LIN {X 0,Y 509.075,Z 406.145,A -85,B 0,C 180,E1 -5489.209,E2 -5489.209} C_VEL
LIN {X 0,Y 509.075,Z 406.145,A -85,B 0,C 180,E1 -5490.791,E2 -5490.791} C_VEL
LIN {X 0,Y 509.114,Z 405.559,A -85,B 0,C 180,E1 -5491.582,E2 -5491.582} C_VEL
LIN {X 0,Y 509.203,Z 403.121,A -85,B 0,C 180,E1 -5493.165,E2 -5493.165} C_VEL
LIN {X 0,Y 509.209,Z 400.177,A -85,B 0,C 180,E1 -5494.353,E2 -5494.353} C_VEL
LIN {X 0,Y 509.293,Z 396.195,A -85,B 0,C 180,E1 -5495.543,E2 -5495.543} C_VEL
LIN {X 0,Y 509.357,Z 391.927,A -85,B 0,C 180,E1 -5496.557,E2 -5496.557} C_VEL
LIN {X 0,Y 509.449,Z 386.963,A -85,B 0,C 180,E1 -5497.53,E2 -5497.53} C_VEL
LIN {X 0,Y 509.619,Z 380.867,A -85,B 0,C 180,E1 -5498.525,E2 -5498.525} C_VEL
LIN {X 0,Y 509.789,Z 375.167,A -85,B 0,C 180,E1 -5499.322,E2 -5499.322} C_VEL
LIN {X 0,Y 510.017,Z 366.61,A -85,B 0,C 180,E1 -5500.319,E2 -5500.319} C_VEL
LIN {X 0,Y 510.299,Z 358.429,A -85,B 0,C 180,E1 -5501.117,E2 -5501.117} C_VEL
LIN {X 0,Y 510.571,Z 349.915,A -85,B 0,C 180,E1 -5501.815,E2 -5501.815} C_VEL
LIN {X 0,Y 510.752,Z 341.423,A -85,B 0,C 180,E1 -5502.401,E2 -5502.401} C_VEL
LIN {X 0,Y 511.054,Z 331.433,A -85,B 0,C 180,E1 -5502.963,E2 -5502.963} C_VEL
LIN {X 0,Y 511.333,Z 321.35,A -85,B 0,C 180,E1 -5503.411,E2 -5503.411} C_VEL
LIN {X 0,Y 511.369,Z 314.018,A -85,B 0,C 180,E1 -5503.676,E2 -5503.676} C_VEL
LIN {X 0,Y 509.54,Z 302.645,A -85,B 0,C 180,E1 -5504.021,E2 -5504.021} C_VEL
LIN {X 0,Y 509.248,Z 300.709,A -85,B 0,C 180,E1 -5504.077,E2 -5504.077} C_VEL
LIN {X 0,Y 509.293,Z 294.675,A -85,B 0,C 180,E1 -5506.845,E2 -5506.845} C_VEL
LIN {X 0,Y 509.362,Z 289.361,A -85,B 0,C 180,E1 -5509.338,E2 -5509.338} C_VEL
LIN {X 0,Y 509.468,Z 282.918,A -85,B 0,C 180,E1 -5512.441,E2 -5512.441} C_VEL
LIN {X 0,Y 509.557,Z 277.151,A -85,B 0,C 180,E1 -5515.312,E2 -5515.312} C_VEL
LIN {X 0,Y 509.71,Z 271.804,A -85,B 0,C 180,E1 -5518.058,E2 -5518.058} C_VEL
LIN {X 0,Y 509.892,Z 266.964,A -85,B 0,C 180,E1 -5520.662,E2 -5520.662} C_VEL
LIN {X 0,Y 510.073,Z 262.008,A -85,B 0,C 180,E1 -5523.444,E2 -5523.444} C_VEL
LIN {X 0,Y 510.239,Z 257.149,A -85,B 0,C 180,E1 -5526.318,E2 -5526.318} C_VEL
LIN {X 0,Y 510.389,Z 252.423,A -85,B 0,C 180,E1 -5529.301,E2 -5529.301} C_VEL
LIN {X 0,Y 510.459,Z 248.462,A -85,B 0,C 180,E1 -5531.969,E2 -5531.969} C_VEL
LIN {X 0,Y 510.205,Z 245.375,A -85,B 0,C 180,E1 -5534.248,E2 -5534.248} C_VEL
LIN {X 0,Y 509.818,Z 242.618,A -85,B 0,C 180,E1 -5536.425,E2 -5536.425} C_VEL
LIN {X 0,Y 509.825,Z 242.479,A -85,B 0,C 180,E1 -5539.302,E2 -5539.302} C_VEL
LIN {X 0,Y 509.853,Z 242.477,A -85,B 0,C 180,E1 -5541.784,E2 -5541.784} C_VEL
LIN {X 0,Y 509.828,Z 242.479,A -85,B 0,C 180,E1 -5544.619,E2 -5544.619} C_VEL
LIN {X 0,Y 509.864,Z 242.471,A -85,B 0,C 180,E1 -5547.478,E2 -5547.478} C_VEL
LIN {X 0,Y 509.861,Z 242.474,A -85,B 0,C 180,E1 -5550.271,E2 -5550.271} C_VEL
LIN {X 0,Y 509.832,Z 242.473,A -85,B 0,C 180,E1 -5552.938,E2 -5552.938} C_VEL
LIN {X 0,Y 509.845,Z 242.476,A -85,B 0,C 180,E1 -5555.569,E2 -5555.569} C_VEL
LIN {X 0,Y 509.821,Z 242.478,A -85,B 0,C 180,E1 -5558.145,E2 -5558.145} C_VEL
LIN {X 0,Y 509.854,Z 242.47,A -85,B 0,C 180,E1 -5560.678,E2 -5560.678} C_VEL
LIN {X 0,Y 509.861,Z 242.472,A -85,B 0,C 180,E1 -5563.17,E2 -5563.17} C_VEL
LIN {X 0,Y 509.857,Z 242.479,A -85,B 0,C 180,E1 -5565.63,E2 -5565.63} C_VEL
LIN {X 0,Y 509.905,Z 242.465,A -85,B 0,C 180,E1 -5568.87,E2 -5568.87} C_VEL
LIN {X 0,Y 509.905,Z 242.465,A -85,B 0,C 180,E1 -5572.074,E2 -5572.074} C_VEL
LIN {X 0,Y 509.959,Z 242.457,A -85,B 0,C 180,E1 -5574.46,E2 -5574.46} C_VEL
LIN {X 0,Y 510.034,Z 242.452,A -85,B 0,C 180,E1 -5577.626,E2 -5577.626} C_VEL
LIN {X 0,Y 510.038,Z 242.448,A -85,B 0,C 180,E1 -5579.995,E2 -5579.995} C_VEL
LIN {X 0,Y 510.035,Z 242.448,A -85,B 0,C 180,E1 -5582.364,E2 -5582.364} C_VEL
LIN {X 0,Y 509.951,Z 242.461,A -85,B 0,C 180,E1 -5585.531,E2 -5585.531} C_VEL
LIN {X 0,Y 509.902,Z 242.464,A -85,B 0,C 180,E1 -5587.917,E2 -5587.917} C_VEL
LIN {X 0,Y 509.895,Z 242.472,A -85,B 0,C 180,E1 -5591.12,E2 -5591.12} C_VEL
LIN {X 0,Y 509.839,Z 242.474,A -85,B 0,C 180,E1 -5594.361,E2 -5594.361} C_VEL
LIN {X 0,Y 509.849,Z 242.48,A -85,B 0,C 180,E1 -5596.821,E2 -5596.821} C_VEL
LIN {X 0,Y 509.889,Z 242.468,A -85,B 0,C 180,E1 -5600.15,E2 -5600.15} C_VEL
LIN {X 0,Y 509.798,Z 242.477,A -85,B 0,C 180,E1 -5603.558,E2 -5603.558} C_VEL
LIN {X 0,Y 509.878,Z 242.473,A -85,B 0,C 180,E1 -5606.373,E2 -5606.373} C_VEL
LIN {X 0,Y 509.841,Z 242.476,A -85,B 0,C 180,E1 -5608.839,E2 -5608.839} C_VEL
LIN {X 0,Y 509.783,Z 242.479,A -85,B 0,C 180,E1 -5611.585,E2 -5611.585} C_VEL
LIN {X 0,Y 509.814,Z 242.484,A -85,B 0,C 180,E1 -5614.408,E2 -5614.408} C_VEL
LIN {X 0,Y 509.776,Z 242.48,A -85,B 0,C 180,E1 -5617.336,E2 -5617.336} C_VEL
LIN {X 0,Y 509.817,Z 242.482,A -85,B 0,C 180,E1 -5620.375,E2 -5620.375} C_VEL
LIN {X 0,Y 509.809,Z 242.476,A -85,B 0,C 180,E1 -5623.062,E2 -5623.062} C_VEL
LIN {X 0,Y 509.781,Z 242.484,A -85,B 0,C 180,E1 -5625.788,E2 -5625.788} C_VEL
LIN {X 0,Y 509.819,Z 242.477,A -85,B 0,C 180,E1 -5628.572,E2 -5628.572} C_VEL
LIN {X 0,Y 509.806,Z 242.481,A -85,B 0,C 180,E1 -5631.659,E2 -5631.659} C_VEL
LIN {X 0,Y 509.776,Z 242.485,A -85,B 0,C 180,E1 -5633.707,E2 -5633.707} C_VEL
LIN {X 0,Y 509.108,Z 242.566,A -85,B 0,C 180,E1 -5634.367,E2 -5634.367} C_VEL
LIN {X 0,Y 506.292,Z 242.917,A -85,B 0,C 180,E1 -5635.439,E2 -5635.439} C_VEL
LIN {X 0,Y 503.9,Z 243.215,A -85,B 0,C 180,E1 -5636.302,E2 -5636.302} C_VEL
LIN {X 0,Y 502.851,Z 243.343,A -85,B 0,C 180,E1 -5636.968,E2 -5636.968} C_VEL
LIN {X 0,Y 502.753,Z 243.355,A -85,B 0,C 180,E1 -5637.194,E2 -5637.194} C_VEL
LIN {X 0,Y 502.771,Z 243.357,A -85,B 0,C 180,E1 -5640.058,E2 -5640.058} C_VEL
LIN {X 0,Y 502.775,Z 243.352,A -85,B 0,C 180,E1 -5642.531,E2 -5642.531} C_VEL
LIN {X 0,Y 502.781,Z 243.356,A -85,B 0,C 180,E1 -5645.292,E2 -5645.292} C_VEL
LIN {X 0,Y 502.757,Z 243.359,A -85,B 0,C 180,E1 -5647.826,E2 -5647.826} C_VEL
LIN {X 0,Y 502.761,Z 243.354,A -85,B 0,C 180,E1 -5650.398,E2 -5650.398} C_VEL
LIN {X 0,Y 502.783,Z 243.356,A -85,B 0,C 180,E1 -5652.93,E2 -5652.93} C_VEL
LIN {X 0,Y 502.796,Z 243.359,A -85,B 0,C 180,E1 -5655.428,E2 -5655.428} C_VEL
LIN {X 0,Y 502.831,Z 243.349,A -85,B 0,C 180,E1 -5658.716,E2 -5658.716} C_VEL
LIN {X 0,Y 502.851,Z 243.346,A -85,B 0,C 180,E1 -5661.966,E2 -5661.966} C_VEL
LIN {X 0,Y 502.899,Z 243.34,A -85,B 0,C 180,E1 -5664.386,E2 -5664.386} C_VEL
LIN {X 0,Y 502.96,Z 243.333,A -85,B 0,C 180,E1 -5667.598,E2 -5667.598} C_VEL
LIN {X 0,Y 502.955,Z 243.333,A -85,B 0,C 180,E1 -5670,E2 -5670} C_VEL
LIN {X 0,Y 502.96,Z 243.333,A -85,B 0,C 180,E1 -5672.402,E2 -5672.402} C_VEL
LIN {X 0,Y 502.899,Z 243.34,A -85,B 0,C 180,E1 -5675.614,E2 -5675.614} C_VEL
LIN {X 0,Y 502.851,Z 243.346,A -85,B 0,C 180,E1 -5678.034,E2 -5678.034} C_VEL
LIN {X 0,Y 502.831,Z 243.349,A -85,B 0,C 180,E1 -5681.284,E2 -5681.284} C_VEL
LIN {X 0,Y 502.796,Z 243.359,A -85,B 0,C 180,E1 -5684.572,E2 -5684.572} C_VEL
LIN {X 0,Y 502.813,Z 243.351,A -85,B 0,C 180,E1 -5687.908,E2 -5687.908} C_VEL
LIN {X 0,Y 502.766,Z 243.362,A -85,B 0,C 180,E1 -5690.539,E2 -5690.539} C_VEL
LIN {X 0,Y 502.759,Z 243.356,A -85,B 0,C 180,E1 -5693.042,E2 -5693.042} C_VEL
LIN {X 0,Y 502.791,Z 243.351,A -85,B 0,C 180,E1 -5695.678,E2 -5695.678} C_VEL
LIN {X 0,Y 502.783,Z 243.359,A -85,B 0,C 180,E1 -5698.375,E2 -5698.375} C_VEL
LIN {X 0,Y 502.737,Z 243.358,A -85,B 0,C 180,E1 -5701.503,E2 -5701.503} C_VEL
LIN {X 0,Y 502.749,Z 243.36,A -85,B 0,C 180,E1 -5704.448,E2 -5704.448} C_VEL
LIN {X 0,Y 502.726,Z 243.358,A -85,B 0,C 180,E1 -5707.182,E2 -5707.182} C_VEL
LIN {X 0,Y 502.79,Z 243.359,A -85,B 0,C 180,E1 -5710.014,E2 -5710.014} C_VEL
LIN {X 0,Y 502.774,Z 243.357,A -85,B 0,C 180,E1 -5712.206,E2 -5712.206} C_VEL
LIN {X 0,Y 502.766,Z 243.359,A -85,B 0,C 180,E1 -5715.669,E2 -5715.669} C_VEL
LIN {X 0,Y 502.783,Z 243.352,A -85,B 0,C 180,E1 -5718.94,E2 -5718.94} C_VEL
LIN {X 0,Y 502.75,Z 243.359,A -85,B 0,C 180,E1 -5722.051,E2 -5722.051} C_VEL
LIN {X 0,Y 502.769,Z 243.354,A -85,B 0,C 180,E1 -5725.04,E2 -5725.04} C_VEL
LIN {X 0,Y 502.746,Z 243.36,A -85,B 0,C 180,E1 -5727.92,E2 -5727.92} C_VEL
LIN {X 0,Y 502.788,Z 243.351,A -85,B 0,C 180,E1 -5730.717,E2 -5730.717} C_VEL
LIN {X 0,Y 502.829,Z 243.354,A -85,B 0,C 180,E1 -5733.444,E2 -5733.444} C_VEL
LIN {X 0,Y 502.753,Z 243.356,A -85,B 0,C 180,E1 -5736.091,E2 -5736.091} C_VEL
LIN {X 0,Y 502.755,Z 243.356,A -85,B 0,C 180,E1 -5738.694,E2 -5738.694} C_VEL
LIN {X 0,Y 502.8,Z 243.358,A -85,B 0,C 180,E1 -5741.253,E2 -5741.253} C_VEL
LIN {X 0,Y 502.825,Z 243.348,A -85,B 0,C 180,E1 -5744.605,E2 -5744.605} C_VEL
LIN {X 0,Y 502.857,Z 243.342,A -85,B 0,C 180,E1 -5748.043,E2 -5748.043} C_VEL
LIN {X 0,Y 502.844,Z 243.35,A -85,B 0,C 180,E1 -5751.161,E2 -5751.161} C_VEL
LIN {X 0,Y 502.876,Z 243.341,A -85,B 0,C 180,E1 -5753.586,E2 -5753.586} C_VEL
LIN {X 0,Y 502.881,Z 243.347,A -85,B 0,C 180,E1 -5756.8,E2 -5756.8} C_VEL
LIN {X 0,Y 502.999,Z 243.327,A -85,B 0,C 180,E1 -5759.204,E2 -5759.204} C_VEL
LIN {X 0,Y 503.023,Z 243.329,A -85,B 0,C 180,E1 -5760.805,E2 -5760.805} C_VEL
LIN {X 0,Y 502.85,Z 243.345,A -85,B 0,C 180,E1 -5763.209,E2 -5763.209} C_VEL
LIN {X 0,Y 502.884,Z 243.345,A -85,B 0,C 180,E1 -5766.424,E2 -5766.424} C_VEL
LIN {X 0,Y 502.842,Z 243.348,A -85,B 0,C 180,E1 -5768.848,E2 -5768.848} C_VEL
LIN {X 0,Y 502.841,Z 243.348,A -85,B 0,C 180,E1 -5772.106,E2 -5772.106} C_VEL
LIN {X 0,Y 502.846,Z 243.343,A -85,B 0,C 180,E1 -5775.404,E2 -5775.404} C_VEL
LIN {X 0,Y 502.82,Z 243.349,A -85,B 0,C 180,E1 -5778.756,E2 -5778.756} C_VEL
LIN {X 0,Y 502.783,Z 243.351,A -85,B 0,C 180,E1 -5781.315,E2 -5781.315} C_VEL
LIN {X 0,Y 502.773,Z 243.358,A -85,B 0,C 180,E1 -5783.918,E2 -5783.918} C_VEL
LIN {X 0,Y 502.791,Z 243.353,A -85,B 0,C 180,E1 -5786.574,E2 -5786.574} C_VEL
LIN {X 0,Y 502.817,Z 243.355,A -85,B 0,C 180,E1 -5789.938,E2 -5789.938} C_VEL
LIN {X 0,Y 502.834,Z 243.345,A -85,B 0,C 180,E1 -5793.034,E2 -5793.034} C_VEL
LIN {X 0,Y 502.771,Z 243.362,A -85,B 0,C 180,E1 -5795.955,E2 -5795.955} C_VEL
LIN {X 0,Y 502.797,Z 243.354,A -85,B 0,C 180,E1 -5798.98,E2 -5798.98} C_VEL
LIN {X 0,Y 502.782,Z 243.359,A -85,B 0,C 180,E1 -5802.198,E2 -5802.198} C_VEL
LIN {X 0,Y 502.785,Z 243.593,A -85,B 0,C 180,E1 -5803.377,E2 -5803.377} C_VEL
LIN {X 0,Y 503.206,Z 246.497,A -85,B 0,C 180,E1 -5805.709,E2 -5805.709} C_VEL
LIN {X 0,Y 503.444,Z 249.486,A -85,B 0,C 180,E1 -5807.929,E2 -5807.929} C_VEL
LIN {X 0,Y 503.39,Z 252.737,A -85,B 0,C 180,E1 -5810.166,E2 -5810.166} C_VEL
LIN {X 0,Y 503.25,Z 257.244,A -85,B 0,C 180,E1 -5813.095,E2 -5813.095} C_VEL
LIN {X 0,Y 503.074,Z 262.087,A -85,B 0,C 180,E1 -5816.028,E2 -5816.028} C_VEL
LIN {X 0,Y 502.875,Z 266.994,A -85,B 0,C 180,E1 -5818.863,E2 -5818.863} C_VEL
LIN {X 0,Y 502.658,Z 272.27,A -85,B 0,C 180,E1 -5821.748,E2 -5821.748} C_VEL
LIN {X 0,Y 502.499,Z 277.115,A -85,B 0,C 180,E1 -5824.306,E2 -5824.306} C_VEL
LIN {X 0,Y 502.397,Z 282.283,A -85,B 0,C 180,E1 -5826.941,E2 -5826.941} C_VEL
LIN {X 0,Y 502.347,Z 287.694,A -85,B 0,C 180,E1 -5829.615,E2 -5829.615} C_VEL
LIN {X 0,Y 502.22,Z 294.546,A -85,B 0,C 180,E1 -5832.911,E2 -5832.911} C_VEL
LIN {X 0,Y 502.173,Z 300.551,A -85,B 0,C 180,E1 -5835.72,E2 -5835.72} C_VEL
LIN {X 0,Y 504.348,Z 314.257,A -85,B 0,C 180,E1 -5836.143,E2 -5836.143} C_VEL
LIN {X 0,Y 504.491,Z 318.58,A -85,B 0,C 180,E1 -5836.301,E2 -5836.301} C_VEL
LIN {X 0,Y 504.215,Z 329.225,A -85,B 0,C 180,E1 -5836.755,E2 -5836.755} C_VEL
LIN {X 0,Y 503.886,Z 338.977,A -85,B 0,C 180,E1 -5837.286,E2 -5837.286} C_VEL
LIN {X 0,Y 503.647,Z 347.066,A -85,B 0,C 180,E1 -5837.82,E2 -5837.82} C_VEL
LIN {X 0,Y 503.385,Z 355.963,A -85,B 0,C 180,E1 -5838.525,E2 -5838.525} C_VEL
LIN {X 0,Y 503.082,Z 364.495,A -85,B 0,C 180,E1 -5839.333,E2 -5839.333} C_VEL
LIN {X 0,Y 502.86,Z 371.717,A -85,B 0,C 180,E1 -5840.142,E2 -5840.142} C_VEL
LIN {X 0,Y 502.657,Z 377.92,A -85,B 0,C 180,E1 -5840.95,E2 -5840.95} C_VEL
LIN {X 0,Y 502.449,Z 384.456,A -85,B 0,C 180,E1 -5841.96,E2 -5841.96} C_VEL
LIN {X 0,Y 502.339,Z 390.012,A -85,B 0,C 180,E1 -5842.989,E2 -5842.989} C_VEL
LIN {X 0,Y 502.217,Z 394.446,A -85,B 0,C 180,E1 -5843.976,E2 -5843.976} C_VEL
LIN {X 0,Y 502.116,Z 398.766,A -85,B 0,C 180,E1 -5845.183,E2 -5845.183} C_VEL
LIN {X 0,Y 502.141,Z 401.131,A -85,B 0,C 180,E1 -5845.987,E2 -5845.987} C_VEL
LIN {X 0,Y 502.123,Z 402.927,A -85,B 0,C 180,E1 -5846.791,E2 -5846.791} C_VEL
LIN {X 0,Y 502.039,Z 405.365,A -85,B 0,C 180,E1 -5848.396,E2 -5848.396} C_VEL
LIN {X 0,Y 501.992,Z 405.95,A -85,B 0,C 180,E1 -5849.198,E2 -5849.198} C_VEL
LIN {X 0,Y 501.992,Z 405.95,A -85,B 0,C 180,E1 -5850.802,E2 -5850.802} C_VEL
LIN {X 0,Y 502.039,Z 405.365,A -85,B 0,C 180,E1 -5851.604,E2 -5851.604} C_VEL
LIN {X 0,Y 502.123,Z 402.927,A -85,B 0,C 180,E1 -5853.209,E2 -5853.209} C_VEL
LIN {X 0,Y 502.107,Z 399.982,A -85,B 0,C 180,E1 -5854.415,E2 -5854.415} C_VEL
LIN {X 0,Y 502.209,Z 396,A -85,B 0,C 180,E1 -5855.622,E2 -5855.622} C_VEL
LIN {X 0,Y 502.284,Z 391.064,A -85,B 0,C 180,E1 -5856.79,E2 -5856.79} C_VEL
LIN {X 0,Y 502.411,Z 385.612,A -85,B 0,C 180,E1 -5857.839,E2 -5857.839} C_VEL
LIN {X 0,Y 502.593,Z 379.295,A -85,B 0,C 180,E1 -5858.848,E2 -5858.848} C_VEL
LIN {X 0,Y 502.813,Z 373.344,A -85,B 0,C 180,E1 -5859.656,E2 -5859.656} C_VEL
LIN {X 0,Y 502.993,Z 366.415,A -85,B 0,C 180,E1 -5860.465,E2 -5860.465} C_VEL
LIN {X 0,Y 503.291,Z 358.233,A -85,B 0,C 180,E1 -5861.273,E2 -5861.273} C_VEL
LIN {X 0,Y 503.572,Z 349.719,A -85,B 0,C 180,E1 -5861.981,E2 -5861.981} C_VEL
LIN {X 0,Y 503.779,Z 341.832,A -85,B 0,C 180,E1 -5862.538,E2 -5862.538} C_VEL
LIN {X 0,Y 504.112,Z 332.246,A -85,B 0,C 180,E1 -5863.094,E2 -5863.094} C_VEL
LIN {X 0,Y 504.411,Z 322.444,A -85,B 0,C 180,E1 -5863.547,E2 -5863.547} C_VEL
LIN {X 0,Y 504.421,Z 314.697,A -85,B 0,C 180,E1 -5863.842,E2 -5863.842} C_VEL
LIN {X 0,Y 502.472,Z 302.766,A -85,B 0,C 180,E1 -5864.216,E2 -5864.216} C_VEL
LIN {X 0,Y 502.173,Z 300.551,A -85,B 0,C 180,E1 -5864.28,E2 -5864.28} C_VEL
LIN {X 0,Y 502.22,Z 294.542,A -85,B 0,C 180,E1 -5867.089,E2 -5867.089} C_VEL
LIN {X 0,Y 502.344,Z 287.506,A -85,B 0,C 180,E1 -5870.472,E2 -5870.472} C_VEL
LIN {X 0,Y 502.397,Z 282.277,A -85,B 0,C 180,E1 -5873.059,E2 -5873.059} C_VEL
LIN {X 0,Y 502.499,Z 277.109,A -85,B 0,C 180,E1 -5875.694,E2 -5875.694} C_VEL
LIN {X 0,Y 502.666,Z 271.992,A -85,B 0,C 180,E1 -5878.383,E2 -5878.383} C_VEL
LIN {X 0,Y 502.877,Z 266.988,A -85,B 0,C 180,E1 -5881.137,E2 -5881.137} C_VEL
LIN {X 0,Y 503.071,Z 262.038,A -85,B 0,C 180,E1 -5883.972,E2 -5883.972} C_VEL
LIN {X 0,Y 503.252,Z 257.233,A -85,B 0,C 180,E1 -5886.905,E2 -5886.905} C_VEL
LIN {X 0,Y 503.392,Z 252.511,A -85,B 0,C 180,E1 -5889.956,E2 -5889.956} C_VEL
LIN {X 0,Y 503.456,Z 249.175,A -85,B 0,C 180,E1 -5892.278,E2 -5892.278} C_VEL
LIN {X 0,Y 503.154,Z 246.143,A -85,B 0,C 180,E1 -5894.57,E2 -5894.57} C_VEL
LIN {X 0,Y 502.763,Z 243.42,A -85,B 0,C 180,E1 -5896.765,E2 -5896.765} C_VEL
LIN {X 0,Y 502.781,Z 243.357,A -85,B 0,C 180,E1 -5899.009,E2 -5899.009} C_VEL
LIN {X 0,Y 502.794,Z 243.358,A -85,B 0,C 180,E1 -5902.043,E2 -5902.043} C_VEL
LIN {X 0,Y 502.797,Z 243.353,A -85,B 0,C 180,E1 -5905.031,E2 -5905.031} C_VEL
LIN {X 0,Y 502.785,Z 243.358,A -85,B 0,C 180,E1 -5907.912,E2 -5907.912} C_VEL
LIN {X 0,Y 502.814,Z 243.348,A -85,B 0,C 180,E1 -5910.708,E2 -5910.708} C_VEL
LIN {X 0,Y 502.791,Z 243.353,A -85,B 0,C 180,E1 -5913.453,E2 -5913.453} C_VEL
LIN {X 0,Y 502.773,Z 243.358,A -85,B 0,C 180,E1 -5916.082,E2 -5916.082} C_VEL
LIN {X 0,Y 502.783,Z 243.351,A -85,B 0,C 180,E1 -5918.685,E2 -5918.685} C_VEL
LIN {X 0,Y 502.82,Z 243.349,A -85,B 0,C 180,E1 -5921.244,E2 -5921.244} C_VEL
LIN {X 0,Y 502.846,Z 243.343,A -85,B 0,C 180,E1 -5924.596,E2 -5924.596} C_VEL
LIN {X 0,Y 502.873,Z 243.342,A -85,B 0,C 180,E1 -5928.035,E2 -5928.035} C_VEL
LIN {X 0,Y 502.842,Z 243.348,A -85,B 0,C 180,E1 -5931.152,E2 -5931.152} C_VEL
LIN {X 0,Y 502.884,Z 243.345,A -85,B 0,C 180,E1 -5933.576,E2 -5933.576} C_VEL
LIN {X 0,Y 502.85,Z 243.345,A -85,B 0,C 180,E1 -5936.791,E2 -5936.791} C_VEL
LIN {X 0,Y 503.023,Z 243.329,A -85,B 0,C 180,E1 -5939.195,E2 -5939.195} C_VEL
LIN {X 0,Y 503.005,Z 243.324,A -85,B 0,C 180,E1 -5942.397,E2 -5942.397} C_VEL
LIN {X 0,Y 502.905,Z 243.338,A -85,B 0,C 180,E1 -5945.609,E2 -5945.609} C_VEL
LIN {X 0,Y 502.862,Z 243.341,A -85,B 0,C 180,E1 -5948.029,E2 -5948.029} C_VEL
LIN {X 0,Y 502.859,Z 243.346,A -85,B 0,C 180,E1 -5951.278,E2 -5951.278} C_VEL
LIN {X 0,Y 502.82,Z 243.351,A -85,B 0,C 180,E1 -5954.566,E2 -5954.566} C_VEL
LIN {X 0,Y 502.796,Z 243.35,A -85,B 0,C 180,E1 -5957.903,E2 -5957.903} C_VEL
LIN {X 0,Y 502.801,Z 243.355,A -85,B 0,C 180,E1 -5960.531,E2 -5960.531} C_VEL
LIN {X 0,Y 502.76,Z 243.358,A -85,B 0,C 180,E1 -5963.035,E2 -5963.035} C_VEL
LIN {X 0,Y 502.806,Z 243.348,A -85,B 0,C 180,E1 -5965.671,E2 -5965.671} C_VEL
LIN {X 0,Y 502.805,Z 243.355,A -85,B 0,C 180,E1 -5968.368,E2 -5968.368} C_VEL
LIN {X 0,Y 502.755,Z 243.355,A -85,B 0,C 180,E1 -5971.494,E2 -5971.494} C_VEL
LIN {X 0,Y 502.766,Z 243.361,A -85,B 0,C 180,E1 -5974.44,E2 -5974.44} C_VEL
LIN {X 0,Y 502.738,Z 243.357,A -85,B 0,C 180,E1 -5977.174,E2 -5977.174} C_VEL
LIN {X 0,Y 502.776,Z 243.357,A -85,B 0,C 180,E1 -5980.007,E2 -5980.007} C_VEL
LIN {X 0,Y 502.782,Z 243.36,A -85,B 0,C 180,E1 -5982.198,E2 -5982.198} C_VEL
LIN {X 0,Y 502.751,Z 243.356,A -85,B 0,C 180,E1 -5985.464,E2 -5985.464} C_VEL
LIN {X 0,Y 502.786,Z 243.357,A -85,B 0,C 180,E1 -5987.861,E2 -5987.861} C_VEL
LIN {X 0,Y 502.775,Z 243.352,A -85,B 0,C 180,E1 -5991.023,E2 -5991.023} C_VEL
LIN {X 0,Y 502.729,Z 243.363,A -85,B 0,C 180,E1 -5994.164,E2 -5994.164} C_VEL
LIN {X 0,Y 502.753,Z 243.355,A -85,B 0,C 180,E1 -5997.194,E2 -5997.194} C_VEL
LIN {X 0,Y 502.053,Z 243.45,A -85,B 0,C 180,E1 -5997.863,E2 -5997.863} C_VEL
LIN {X 0,Y 499.195,Z 243.8,A -85,B 0,C 180,E1 -5998.949,E2 -5998.949} C_VEL
LIN {X 0,Y 496.804,Z 244.104,A -85,B 0,C 180,E1 -5999.824,E2 -5999.824} C_VEL
LIN {X 0,Y 495.785,Z 244.224,A -85,B 0,C 180,E1 -6000.5,E2 -6000.5} C_VEL
LIN {X 0,Y 495.705,Z 244.233,A -85,B 0,C 180,E1 -6000.728,E2 -6000.728} C_VEL
LIN {X 0,Y 495.744,Z 244.233,A -85,B 0,C 180,E1 -6003.93,E2 -6003.93} C_VEL
LIN {X 0,Y 495.726,Z 244.233,A -85,B 0,C 180,E1 -6007.128,E2 -6007.128} C_VEL
LIN {X 0,Y 495.713,Z 244.234,A -85,B 0,C 180,E1 -6010.108,E2 -6010.108} C_VEL
LIN {X 0,Y 495.736,Z 244.232,A -85,B 0,C 180,E1 -6012.68,E2 -6012.68} C_VEL
LIN {X 0,Y 495.749,Z 244.235,A -85,B 0,C 180,E1 -6015.216,E2 -6015.216} C_VEL
LIN {X 0,Y 495.81,Z 244.222,A -85,B 0,C 180,E1 -6018.554,E2 -6018.554} C_VEL
LIN {X 0,Y 495.819,Z 244.223,A -85,B 0,C 180,E1 -6021.851,E2 -6021.851} C_VEL
LIN {X 0,Y 495.854,Z 244.217,A -85,B 0,C 180,E1 -6024.306,E2 -6024.306} C_VEL
LIN {X 0,Y 495.93,Z 244.209,A -85,B 0,C 180,E1 -6027.563,E2 -6027.563} C_VEL
LIN {X 0,Y 495.926,Z 244.209,A -85,B 0,C 180,E1 -6030,E2 -6030} C_VEL
LIN {X 0,Y 495.93,Z 244.209,A -85,B 0,C 180,E1 -6032.437,E2 -6032.437} C_VEL
LIN {X 0,Y 495.854,Z 244.217,A -85,B 0,C 180,E1 -6035.694,E2 -6035.694} C_VEL
LIN {X 0,Y 495.819,Z 244.223,A -85,B 0,C 180,E1 -6038.149,E2 -6038.149} C_VEL
LIN {X 0,Y 495.81,Z 244.222,A -85,B 0,C 180,E1 -6041.446,E2 -6041.446} C_VEL
LIN {X 0,Y 495.749,Z 244.235,A -85,B 0,C 180,E1 -6044.784,E2 -6044.784} C_VEL
LIN {X 0,Y 495.765,Z 244.232,A -85,B 0,C 180,E1 -6048.258,E2 -6048.258} C_VEL
LIN {X 0,Y 495.702,Z 244.234,A -85,B 0,C 180,E1 -6051.63,E2 -6051.63} C_VEL
LIN {X 0,Y 495.745,Z 244.23,A -85,B 0,C 180,E1 -6054.884,E2 -6054.884} C_VEL
LIN {X 0,Y 495.759,Z 244.227,A -85,B 0,C 180,E1 -6056.977,E2 -6056.977} C_VEL
LIN {X 0,Y 495.717,Z 244.239,A -85,B 0,C 180,E1 -6060.153,E2 -6060.153} C_VEL
LIN {X 0,Y 495.735,Z 244.229,A -85,B 0,C 180,E1 -6063.248,E2 -6063.248} C_VEL
LIN {X 0,Y 495.672,Z 244.246,A -85,B 0,C 180,E1 -6066.094,E2 -6066.094} C_VEL
LIN {X 0,Y 495.732,Z 244.23,A -85,B 0,C 180,E1 -6068.776,E2 -6068.776} C_VEL
LIN {X 0,Y 495.733,Z 244.235,A -85,B 0,C 180,E1 -6071.782,E2 -6071.782} C_VEL
LIN {X 0,Y 495.709,Z 244.233,A -85,B 0,C 180,E1 -6075.143,E2 -6075.143} C_VEL
LIN {X 0,Y 495.739,Z 244.232,A -85,B 0,C 180,E1 -6078.227,E2 -6078.227} C_VEL
LIN {X 0,Y 495.724,Z 244.233,A -85,B 0,C 180,E1 -6081.236,E2 -6081.236} C_VEL
LIN {X 0,Y 495.716,Z 244.232,A -85,B 0,C 180,E1 -6084.468,E2 -6084.468} C_VEL
LIN {X 0,Y 495.729,Z 244.236,A -85,B 0,C 180,E1 -6087.411,E2 -6087.411} C_VEL
LIN {X 0,Y 495.73,Z 244.23,A -85,B 0,C 180,E1 -6090.259,E2 -6090.259} C_VEL
LIN {X 0,Y 495.79,Z 244.229,A -85,B 0,C 180,E1 -6093.256,E2 -6093.256} C_VEL
LIN {X 0,Y 495.716,Z 244.235,A -85,B 0,C 180,E1 -6095.73,E2 -6095.73} C_VEL
LIN {X 0,Y 495.713,Z 244.232,A -85,B 0,C 180,E1 -6098.376,E2 -6098.376} C_VEL
LIN {X 0,Y 495.756,Z 244.232,A -85,B 0,C 180,E1 -6100.977,E2 -6100.977} C_VEL
LIN {X 0,Y 495.783,Z 244.224,A -85,B 0,C 180,E1 -6104.381,E2 -6104.381} C_VEL
LIN {X 0,Y 495.76,Z 244.232,A -85,B 0,C 180,E1 -6106.896,E2 -6106.896} C_VEL
LIN {X 0,Y 495.755,Z 244.23,A -85,B 0,C 180,E1 -6109.386,E2 -6109.386} C_VEL
LIN {X 0,Y 495.818,Z 244.219,A -85,B 0,C 180,E1 -6111.856,E2 -6111.856} C_VEL
LIN {X 0,Y 495.861,Z 244.215,A -85,B 0,C 180,E1 -6114.311,E2 -6114.311} C_VEL
LIN {X 0,Y 495.975,Z 244.2,A -85,B 0,C 180,E1 -6117.569,E2 -6117.569} C_VEL
LIN {X 0,Y 495.972,Z 244.207,A -85,B 0,C 180,E1 -6120.817,E2 -6120.817} C_VEL
LIN {X 0,Y 495.971,Z 244.205,A -85,B 0,C 180,E1 -6122.441,E2 -6122.441} C_VEL
LIN {X 0,Y 495.87,Z 244.213,A -85,B 0,C 180,E1 -6125.698,E2 -6125.698} C_VEL
LIN {X 0,Y 495.822,Z 244.222,A -85,B 0,C 180,E1 -6128.153,E2 -6128.153} C_VEL
LIN {X 0,Y 495.846,Z 244.215,A -85,B 0,C 180,E1 -6131.449,E2 -6131.449} C_VEL
LIN {X 0,Y 495.785,Z 244.226,A -85,B 0,C 180,E1 -6134.787,E2 -6134.787} C_VEL
LIN {X 0,Y 495.778,Z 244.231,A -85,B 0,C 180,E1 -6138.175,E2 -6138.175} C_VEL
LIN {X 0,Y 495.775,Z 244.226,A -85,B 0,C 180,E1 -6140.76,E2 -6140.76} C_VEL
LIN {X 0,Y 495.742,Z 244.229,A -85,B 0,C 180,E1 -6143.391,E2 -6143.391} C_VEL
LIN {X 0,Y 495.745,Z 244.229,A -85,B 0,C 180,E1 -6146.734,E2 -6146.734} C_VEL
LIN {X 0,Y 495.765,Z 244.23,A -85,B 0,C 180,E1 -6149.75,E2 -6149.75} C_VEL
LIN {X 0,Y 495.77,Z 244.226,A -85,B 0,C 180,E1 -6152.598,E2 -6152.598} C_VEL
LIN {X 0,Y 495.747,Z 244.232,A -85,B 0,C 180,E1 -6155.541,E2 -6155.541} C_VEL
LIN {X 0,Y 495.762,Z 244.23,A -85,B 0,C 180,E1 -6158.77,E2 -6158.77} C_VEL
LIN {X 0,Y 495.751,Z 244.236,A -85,B 0,C 180,E1 -6161.785,E2 -6161.785} C_VEL
LIN {X 0,Y 495.715,Z 244.239,A -85,B 0,C 180,E1 -6162.887,E2 -6162.887} C_VEL
LIN {X 0,Y 496.27,Z 248.129,A -85,B 0,C 180,E1 -6166.06,E2 -6166.06} C_VEL
LIN {X 0,Y 496.448,Z 251.591,A -85,B 0,C 180,E1 -6168.619,E2 -6168.619} C_VEL
LIN {X 0,Y 496.294,Z 255.743,A -85,B 0,C 180,E1 -6171.46,E2 -6171.46} C_VEL
LIN {X 0,Y 496.135,Z 260.505,A -85,B 0,C 180,E1 -6174.495,E2 -6174.495} C_VEL
LIN {X 0,Y 495.928,Z 265.372,A -85,B 0,C 180,E1 -6177.418,E2 -6177.418} C_VEL
LIN {X 0,Y 495.731,Z 270.324,A -85,B 0,C 180,E1 -6180.252,E2 -6180.252} C_VEL
LIN {X 0,Y 495.517,Z 275.965,A -85,B 0,C 180,E1 -6183.325,E2 -6183.325} C_VEL
LIN {X 0,Y 495.387,Z 280.503,A -85,B 0,C 180,E1 -6185.707,E2 -6185.707} C_VEL
LIN {X 0,Y 495.278,Z 285.676,A -85,B 0,C 180,E1 -6188.35,E2 -6188.35} C_VEL
LIN {X 0,Y 495.178,Z 290.91,A -85,B 0,C 180,E1 -6190.948,E2 -6190.948} C_VEL
LIN {X 0,Y 495.104,Z 296.196,A -85,B 0,C 180,E1 -6193.507,E2 -6193.507} C_VEL
LIN {X 0,Y 495.063,Z 300.421,A -85,B 0,C 180,E1 -6195.524,E2 -6195.524} C_VEL
LIN {X 0,Y 496.766,Z 310.981,A -85,B 0,C 180,E1 -6195.836,E2 -6195.836} C_VEL
LIN {X 0,Y 497.647,Z 317.097,A -85,B 0,C 180,E1 -6196.057,E2 -6196.057} C_VEL
LIN {X 0,Y 497.316,Z 328.022,A -85,B 0,C 180,E1 -6196.516,E2 -6196.516} C_VEL
LIN {X 0,Y 496.94,Z 339.052,A -85,B 0,C 180,E1 -6197.122,E2 -6197.122} C_VEL
LIN {X 0,Y 496.632,Z 348.171,A -85,B 0,C 180,E1 -6197.745,E2 -6197.745} C_VEL
LIN {X 0,Y 496.361,Z 356.903,A -85,B 0,C 180,E1 -6198.464,E2 -6198.464} C_VEL
LIN {X 0,Y 496.09,Z 364.3,A -85,B 0,C 180,E1 -6199.181,E2 -6199.181} C_VEL
LIN {X 0,Y 495.83,Z 371.521,A -85,B 0,C 180,E1 -6200.001,E2 -6200.001} C_VEL
LIN {X 0,Y 495.624,Z 377.724,A -85,B 0,C 180,E1 -6200.821,E2 -6200.821} C_VEL
LIN {X 0,Y 495.394,Z 384.261,A -85,B 0,C 180,E1 -6201.844,E2 -6201.844} C_VEL
LIN {X 0,Y 495.275,Z 388.762,A -85,B 0,C 180,E1 -6202.663,E2 -6202.663} C_VEL
LIN {X 0,Y 495.13,Z 393.772,A -85,B 0,C 180,E1 -6203.763,E2 -6203.763} C_VEL
LIN {X 0,Y 495.11,Z 397.334,A -85,B 0,C 180,E1 -6204.706,E2 -6204.706} C_VEL
LIN {X 0,Y 495.035,Z 400.936,A -85,B 0,C 180,E1 -6205.93,E2 -6205.93} C_VEL
LIN {X 0,Y 495.045,Z 402.732,A -85,B 0,C 180,E1 -6206.745,E2 -6206.745} C_VEL
LIN {X 0,Y 494.965,Z 405.171,A -85,B 0,C 180,E1 -6208.373,E2 -6208.373} C_VEL
LIN {X 0,Y 494.913,Z 405.756,A -85,B 0,C 180,E1 -6209.186,E2 -6209.186} C_VEL
LIN {X 0,Y 494.913,Z 405.756,A -85,B 0,C 180,E1 -6210.814,E2 -6210.814} C_VEL
LIN {X 0,Y 494.965,Z 405.171,A -85,B 0,C 180,E1 -6211.627,E2 -6211.627} C_VEL
LIN {X 0,Y 495.045,Z 402.732,A -85,B 0,C 180,E1 -6213.255,E2 -6213.255} C_VEL
LIN {X 0,Y 495.014,Z 399.787,A -85,B 0,C 180,E1 -6214.478,E2 -6214.478} C_VEL
LIN {X 0,Y 495.126,Z 395.804,A -85,B 0,C 180,E1 -6215.702,E2 -6215.702} C_VEL
LIN {X 0,Y 495.226,Z 390.678,A -85,B 0,C 180,E1 -6216.928,E2 -6216.928} C_VEL
LIN {X 0,Y 495.352,Z 385.416,A -85,B 0,C 180,E1 -6217.951,E2 -6217.951} C_VEL
LIN {X 0,Y 495.566,Z 379.1,A -85,B 0,C 180,E1 -6218.975,E2 -6218.975} C_VEL
LIN {X 0,Y 495.764,Z 373.148,A -85,B 0,C 180,E1 -6219.794,E2 -6219.794} C_VEL
LIN {X 0,Y 495.987,Z 366.219,A -85,B 0,C 180,E1 -6220.615,E2 -6220.615} C_VEL
LIN {X 0,Y 496.317,Z 358.038,A -85,B 0,C 180,E1 -6221.434,E2 -6221.434} C_VEL
LIN {X 0,Y 496.606,Z 349.524,A -85,B 0,C 180,E1 -6222.152,E2 -6222.152} C_VEL
LIN {X 0,Y 496.886,Z 340.643,A -85,B 0,C 180,E1 -6222.778,E2 -6222.778} C_VEL
LIN {X 0,Y 497.151,Z 331.042,A -85,B 0,C 180,E1 -6223.332,E2 -6223.332} C_VEL
LIN {X 0,Y 497.493,Z 322.249,A -85,B 0,C 180,E1 -6223.739,E2 -6223.739} C_VEL
LIN {X 0,Y 497.466,Z 315.346,A -85,B 0,C 180,E1 -6224.013,E2 -6224.013} C_VEL
LIN {X 0,Y 495.411,Z 302.577,A -85,B 0,C 180,E1 -6224.423,E2 -6224.423} C_VEL
LIN {X 0,Y 495.049,Z 300.392,A -85,B 0,C 180,E1 -6224.49,E2 -6224.49} C_VEL
LIN {X 0,Y 495.162,Z 294.41,A -85,B 0,C 180,E1 -6227.341,E2 -6227.341} C_VEL
LIN {X 0,Y 495.256,Z 287.407,A -85,B 0,C 180,E1 -6230.779,E2 -6230.779} C_VEL
LIN {X 0,Y 495.327,Z 282.205,A -85,B 0,C 180,E1 -6233.408,E2 -6233.408} C_VEL
LIN {X 0,Y 495.452,Z 277.066,A -85,B 0,C 180,E1 -6236.086,E2 -6236.086} C_VEL
LIN {X 0,Y 495.649,Z 271.992,A -85,B 0,C 180,E1 -6238.822,E2 -6238.822} C_VEL
LIN {X 0,Y 495.871,Z 266.785,A -85,B 0,C 180,E1 -6241.743,E2 -6241.743} C_VEL
LIN {X 0,Y 496.079,Z 261.723,A -85,B 0,C 180,E1 -6244.742,E2 -6244.742} C_VEL
LIN {X 0,Y 496.271,Z 257.28,A -85,B 0,C 180,E1 -6247.525,E2 -6247.525} C_VEL
LIN {X 0,Y 496.398,Z 252.625,A -85,B 0,C 180,E1 -6250.636,E2 -6250.636} C_VEL
LIN {X 0,Y 496.4,Z 249.605,A -85,B 0,C 180,E1 -6252.81,E2 -6252.81} C_VEL
LIN {X 0,Y 496.062,Z 246.645,A -85,B 0,C 180,E1 -6255.102,E2 -6255.102} C_VEL
LIN {X 0,Y 495.715,Z 244.239,A -85,B 0,C 180,E1 -6257.113,E2 -6257.113} C_VEL
LIN {X 0,Y 495.75,Z 244.235,A -85,B 0,C 180,E1 -6259.953,E2 -6259.953} C_VEL
LIN {X 0,Y 495.722,Z 244.238,A -85,B 0,C 180,E1 -6262.552,E2 -6262.552} C_VEL
LIN {X 0,Y 495.774,Z 244.229,A -85,B 0,C 180,E1 -6265.453,E2 -6265.453} C_VEL
LIN {X 0,Y 495.757,Z 244.23,A -85,B 0,C 180,E1 -6268.361,E2 -6268.361} C_VEL
LIN {X 0,Y 495.735,Z 244.23,A -85,B 0,C 180,E1 -6271.179,E2 -6271.179} C_VEL
LIN {X 0,Y 495.733,Z 244.238,A -85,B 0,C 180,E1 -6273.925,E2 -6273.925} C_VEL
LIN {X 0,Y 495.759,Z 244.227,A -85,B 0,C 180,E1 -6277.136,E2 -6277.136} C_VEL
LIN {X 0,Y 495.767,Z 244.229,A -85,B 0,C 180,E1 -6280.106,E2 -6280.106} C_VEL
LIN {X 0,Y 495.754,Z 244.227,A -85,B 0,C 180,E1 -6282.676,E2 -6282.676} C_VEL
LIN {X 0,Y 495.785,Z 244.226,A -85,B 0,C 180,E1 -6285.213,E2 -6285.213} C_VEL
LIN {X 0,Y 495.845,Z 244.215,A -85,B 0,C 180,E1 -6288.551,E2 -6288.551} C_VEL
LIN {X 0,Y 495.822,Z 244.221,A -85,B 0,C 180,E1 -6291.847,E2 -6291.847} C_VEL
LIN {X 0,Y 495.87,Z 244.213,A -85,B 0,C 180,E1 -6294.302,E2 -6294.302} C_VEL
LIN {X 0,Y 495.971,Z 244.205,A -85,B 0,C 180,E1 -6297.559,E2 -6297.559} C_VEL
LIN {X 0,Y 495.981,Z 244.199,A -85,B 0,C 180,E1 -6299.995,E2 -6299.995} C_VEL
LIN {X 0,Y 495.975,Z 244.2,A -85,B 0,C 180,E1 -6302.431,E2 -6302.431} C_VEL
LIN {X 0,Y 495.861,Z 244.215,A -85,B 0,C 180,E1 -6305.689,E2 -6305.689} C_VEL
LIN {X 0,Y 495.818,Z 244.219,A -85,B 0,C 180,E1 -6308.144,E2 -6308.144} C_VEL
LIN {X 0,Y 495.833,Z 244.219,A -85,B 0,C 180,E1 -6311.44,E2 -6311.44} C_VEL
LIN {X 0,Y 495.766,Z 244.233,A -85,B 0,C 180,E1 -6314.778,E2 -6314.778} C_VEL
LIN {X 0,Y 495.739,Z 244.231,A -85,B 0,C 180,E1 -6317.314,E2 -6317.314} C_VEL
LIN {X 0,Y 495.743,Z 244.228,A -85,B 0,C 180,E1 -6319.885,E2 -6319.885} C_VEL
LIN {X 0,Y 495.729,Z 244.236,A -85,B 0,C 180,E1 -6322.855,E2 -6322.855} C_VEL
LIN {X 0,Y 495.757,Z 244.229,A -85,B 0,C 180,E1 -6326.063,E2 -6326.063} C_VEL
LIN {X 0,Y 495.737,Z 244.234,A -85,B 0,C 180,E1 -6328.81,E2 -6328.81} C_VEL
LIN {X 0,Y 495.717,Z 244.232,A -85,B 0,C 180,E1 -6331.72,E2 -6331.72} C_VEL
LIN {X 0,Y 495.736,Z 244.233,A -85,B 0,C 180,E1 -6334.69,E2 -6334.69} C_VEL
LIN {X 0,Y 495.688,Z 244.236,A -85,B 0,C 180,E1 -6337.557,E2 -6337.557} C_VEL
LIN {X 0,Y 495.735,Z 244.232,A -85,B 0,C 180,E1 -6340.694,E2 -6340.694} C_VEL
LIN {X 0,Y 495.728,Z 244.233,A -85,B 0,C 180,E1 -6343.696,E2 -6343.696} C_VEL
LIN {X 0,Y 495.712,Z 244.232,A -85,B 0,C 180,E1 -6347.117,E2 -6347.117} C_VEL
LIN {X 0,Y 495.749,Z 244.231,A -85,B 0,C 180,E1 -6350.363,E2 -6350.363} C_VEL
LIN {X 0,Y 495.677,Z 244.239,A -85,B 0,C 180,E1 -6353.453,E2 -6353.453} C_VEL
LIN {X 0,Y 495.703,Z 244.235,A -85,B 0,C 180,E1 -6356.432,E2 -6356.432} C_VEL
LIN {X 0,Y 495.697,Z 244.237,A -85,B 0,C 180,E1 -6359.31,E2 -6359.31} C_VEL
LIN {X 0,Y 495.705,Z 244.233,A -85,B 0,C 180,E1 -6360.728,E2 -6360.728} C_VEL
LIN {X 0,Y 495.043,Z 244.322,A -85,B 0,C 180,E1 -6361.407,E2 -6361.407} C_VEL
LIN {X 0,Y 492.187,Z 244.673,A -85,B 0,C 180,E1 -6362.51,E2 -6362.51} C_VEL
LIN {X 0,Y 489.78,Z 244.976,A -85,B 0,C 180,E1 -6363.399,E2 -6363.399} C_VEL
LIN {X 0,Y 488.764,Z 245.1,A -85,B 0,C 180,E1 -6364.085,E2 -6364.085} C_VEL
LIN {X 0,Y 488.69,Z 245.107,A -85,B 0,C 180,E1 -6364.318,E2 -6364.318} C_VEL
LIN {X 0,Y 488.688,Z 245.11,A -85,B 0,C 180,E1 -6367.152,E2 -6367.152} C_VEL
LIN {X 0,Y 488.664,Z 245.116,A -85,B 0,C 180,E1 -6369.808,E2 -6369.808} C_VEL
LIN {X 0,Y 488.684,Z 245.11,A -85,B 0,C 180,E1 -6372.422,E2 -6372.422} C_VEL
LIN {X 0,Y 488.72,Z 245.109,A -85,B 0,C 180,E1 -6374.999,E2 -6374.999} C_VEL
LIN {X 0,Y 488.767,Z 245.099,A -85,B 0,C 180,E1 -6378.387,E2 -6378.387} C_VEL
LIN {X 0,Y 488.782,Z 245.1,A -85,B 0,C 180,E1 -6381.733,E2 -6381.733} C_VEL
LIN {X 0,Y 488.811,Z 245.095,A -85,B 0,C 180,E1 -6384.224,E2 -6384.224} C_VEL
LIN {X 0,Y 488.899,Z 245.086,A -85,B 0,C 180,E1 -6387.528,E2 -6387.528} C_VEL
LIN {X 0,Y 488.898,Z 245.085,A -85,B 0,C 180,E1 -6390,E2 -6390} C_VEL
LIN {X 0,Y 488.899,Z 245.086,A -85,B 0,C 180,E1 -6392.472,E2 -6392.472} C_VEL
LIN {X 0,Y 488.811,Z 245.095,A -85,B 0,C 180,E1 -6395.776,E2 -6395.776} C_VEL
LIN {X 0,Y 488.782,Z 245.1,A -85,B 0,C 180,E1 -6398.267,E2 -6398.267} C_VEL
LIN {X 0,Y 488.767,Z 245.099,A -85,B 0,C 180,E1 -6401.613,E2 -6401.613} C_VEL
LIN {X 0,Y 488.72,Z 245.109,A -85,B 0,C 180,E1 -6405.001,E2 -6405.001} C_VEL
LIN {X 0,Y 488.702,Z 245.113,A -85,B 0,C 180,E1 -6408.444,E2 -6408.444} C_VEL
LIN {X 0,Y 488.678,Z 245.11,A -85,B 0,C 180,E1 -6411.071,E2 -6411.071} C_VEL
LIN {X 0,Y 488.655,Z 245.112,A -85,B 0,C 180,E1 -6413.747,E2 -6413.747} C_VEL
LIN {X 0,Y 488.737,Z 245.102,A -85,B 0,C 180,E1 -6416.948,E2 -6416.948} C_VEL
LIN {X 0,Y 488.659,Z 245.118,A -85,B 0,C 180,E1 -6420.368,E2 -6420.368} C_VEL
LIN {X 0,Y 488.678,Z 245.109,A -85,B 0,C 180,E1 -6423.488,E2 -6423.488} C_VEL
LIN {X 0,Y 488.633,Z 245.119,A -85,B 0,C 180,E1 -6426.36,E2 -6426.36} C_VEL
LIN {X 0,Y 488.704,Z 245.106,A -85,B 0,C 180,E1 -6429.253,E2 -6429.253} C_VEL
LIN {X 0,Y 488.682,Z 245.11,A -85,B 0,C 180,E1 -6432.525,E2 -6432.525} C_VEL
LIN {X 0,Y 488.691,Z 245.114,A -85,B 0,C 180,E1 -6435.976,E2 -6435.976} C_VEL
LIN {X 0,Y 488.681,Z 245.108,A -85,B 0,C 180,E1 -6438.591,E2 -6438.591} C_VEL
LIN {X 0,Y 488.696,Z 245.107,A -85,B 0,C 180,E1 -6440.947,E2 -6440.947} C_VEL
LIN {X 0,Y 488.644,Z 245.118,A -85,B 0,C 180,E1 -6443.874,E2 -6443.874} C_VEL
LIN {X 0,Y 488.7,Z 245.106,A -85,B 0,C 180,E1 -6446.882,E2 -6446.882} C_VEL
LIN {X 0,Y 488.687,Z 245.112,A -85,B 0,C 180,E1 -6449.786,E2 -6449.786} C_VEL
LIN {X 0,Y 488.758,Z 245.102,A -85,B 0,C 180,E1 -6453.062,E2 -6453.062} C_VEL
LIN {X 0,Y 488.657,Z 245.111,A -85,B 0,C 180,E1 -6456.26,E2 -6456.26} C_VEL
LIN {X 0,Y 488.718,Z 245.111,A -85,B 0,C 180,E1 -6459.181,E2 -6459.181} C_VEL
LIN {X 0,Y 488.723,Z 245.106,A -85,B 0,C 180,E1 -6461.637,E2 -6461.637} C_VEL
LIN {X 0,Y 488.738,Z 245.108,A -85,B 0,C 180,E1 -6465.005,E2 -6465.005} C_VEL
LIN {X 0,Y 488.787,Z 245.096,A -85,B 0,C 180,E1 -6468.393,E2 -6468.393} C_VEL
LIN {X 0,Y 488.766,Z 245.098,A -85,B 0,C 180,E1 -6471.738,E2 -6471.738} C_VEL
LIN {X 0,Y 488.82,Z 245.092,A -85,B 0,C 180,E1 -6474.229,E2 -6474.229} C_VEL
LIN {X 0,Y 488.943,Z 245.076,A -85,B 0,C 180,E1 -6477.534,E2 -6477.534} C_VEL
LIN {X 0,Y 488.923,Z 245.085,A -85,B 0,C 180,E1 -6480.828,E2 -6480.828} C_VEL
LIN {X 0,Y 488.938,Z 245.081,A -85,B 0,C 180,E1 -6482.476,E2 -6482.476} C_VEL
LIN {X 0,Y 488.828,Z 245.09,A -85,B 0,C 180,E1 -6485.781,E2 -6485.781} C_VEL
LIN {X 0,Y 488.768,Z 245.102,A -85,B 0,C 180,E1 -6488.272,E2 -6488.272} C_VEL
LIN {X 0,Y 488.8,Z 245.093,A -85,B 0,C 180,E1 -6491.617,E2 -6491.617} C_VEL
LIN {X 0,Y 488.758,Z 245.1,A -85,B 0,C 180,E1 -6495.005,E2 -6495.005} C_VEL
LIN {X 0,Y 488.745,Z 245.107,A -85,B 0,C 180,E1 -6498.446,E2 -6498.446} C_VEL
LIN {X 0,Y 488.707,Z 245.105,A -85,B 0,C 180,E1 -6501.074,E2 -6501.074} C_VEL
LIN {X 0,Y 488.674,Z 245.112,A -85,B 0,C 180,E1 -6503.75,E2 -6503.75} C_VEL
LIN {X 0,Y 488.703,Z 245.105,A -85,B 0,C 180,E1 -6506.926,E2 -6506.926} C_VEL
LIN {X 0,Y 488.725,Z 245.108,A -85,B 0,C 180,E1 -6510.223,E2 -6510.223} C_VEL
LIN {X 0,Y 488.735,Z 245.104,A -85,B 0,C 180,E1 -6513.486,E2 -6513.486} C_VEL
LIN {X 0,Y 488.677,Z 245.114,A -85,B 0,C 180,E1 -6516.355,E2 -6516.355} C_VEL
LIN {X 0,Y 488.698,Z 245.112,A -85,B 0,C 180,E1 -6519.258,E2 -6519.258} C_VEL
LIN {X 0,Y 488.677,Z 245.116,A -85,B 0,C 180,E1 -6522.53,E2 -6522.53} C_VEL
LIN {X 0,Y 489.137,Z 248.282,A -85,B 0,C 180,E1 -6525.249,E2 -6525.249} C_VEL
LIN {X 0,Y 489.429,Z 251.23,A -85,B 0,C 180,E1 -6527.555,E2 -6527.555} C_VEL
LIN {X 0,Y 489.363,Z 254.277,A -85,B 0,C 180,E1 -6529.74,E2 -6529.74} C_VEL
LIN {X 0,Y 489.248,Z 257.917,A -85,B 0,C 180,E1 -6532.195,E2 -6532.195} C_VEL
LIN {X 0,Y 489.063,Z 262.279,A -85,B 0,C 180,E1 -6534.999,E2 -6534.999} C_VEL
LIN {X 0,Y 488.851,Z 267.298,A -85,B 0,C 180,E1 -6538.022,E2 -6538.022} C_VEL
LIN {X 0,Y 488.618,Z 271.992,A -85,B 0,C 180,E1 -6540.724,E2 -6540.724} C_VEL
LIN {X 0,Y 488.431,Z 277.033,A -85,B 0,C 180,E1 -6543.51,E2 -6543.51} C_VEL
LIN {X 0,Y 488.279,Z 282.146,A -85,B 0,C 180,E1 -6546.234,E2 -6546.234} C_VEL
LIN {X 0,Y 488.179,Z 288.205,A -85,B 0,C 180,E1 -6549.356,E2 -6549.356} C_VEL
LIN {X 0,Y 488.074,Z 294.278,A -85,B 0,C 180,E1 -6552.399,E2 -6552.399} C_VEL
LIN {X 0,Y 488.01,Z 300.264,A -85,B 0,C 180,E1 -6555.31,E2 -6555.31} C_VEL
LIN {X 0,Y 489.693,Z 310.781,A -85,B 0,C 180,E1 -6555.627,E2 -6555.627} C_VEL
LIN {X 0,Y 490.703,Z 318.19,A -85,B 0,C 180,E1 -6555.908,E2 -6555.908} C_VEL
LIN {X 0,Y 490.373,Z 328.834,A -85,B 0,C 180,E1 -6556.374,E2 -6556.374} C_VEL
LIN {X 0,Y 489.997,Z 338.98,A -85,B 0,C 180,E1 -6556.945,E2 -6556.945} C_VEL
LIN {X 0,Y 489.654,Z 347.975,A -85,B 0,C 180,E1 -6557.567,E2 -6557.567} C_VEL
LIN {X 0,Y 489.382,Z 356.708,A -85,B 0,C 180,E1 -6558.297,E2 -6558.297} C_VEL
LIN {X 0,Y 489.105,Z 364.105,A -85,B 0,C 180,E1 -6559.025,E2 -6559.025} C_VEL
LIN {X 0,Y 488.799,Z 371.325,A -85,B 0,C 180,E1 -6559.856,E2 -6559.856} C_VEL
LIN {X 0,Y 488.565,Z 377.528,A -85,B 0,C 180,E1 -6560.687,E2 -6560.687} C_VEL
LIN {X 0,Y 488.328,Z 384.065,A -85,B 0,C 180,E1 -6561.725,E2 -6561.725} C_VEL
LIN {X 0,Y 488.204,Z 388.567,A -85,B 0,C 180,E1 -6562.556,E2 -6562.556} C_VEL
LIN {X 0,Y 488.029,Z 394.04,A -85,B 0,C 180,E1 -6563.796,E2 -6563.796} C_VEL
LIN {X 0,Y 487.973,Z 398.377,A -85,B 0,C 180,E1 -6565.043,E2 -6565.043} C_VEL
LIN {X 0,Y 487.931,Z 400.741,A -85,B 0,C 180,E1 -6565.87,E2 -6565.87} C_VEL
LIN {X 0,Y 487.968,Z 402.538,A -85,B 0,C 180,E1 -6566.697,E2 -6566.697} C_VEL
LIN {X 0,Y 487.894,Z 404.977,A -85,B 0,C 180,E1 -6568.349,E2 -6568.349} C_VEL
LIN {X 0,Y 487.836,Z 405.562,A -85,B 0,C 180,E1 -6569.175,E2 -6569.175} C_VEL
LIN {X 0,Y 487.836,Z 405.562,A -85,B 0,C 180,E1 -6570.825,E2 -6570.825} C_VEL
LIN {X 0,Y 487.894,Z 404.977,A -85,B 0,C 180,E1 -6571.651,E2 -6571.651} C_VEL
LIN {X 0,Y 487.968,Z 402.538,A -85,B 0,C 180,E1 -6573.303,E2 -6573.303} C_VEL
LIN {X 0,Y 487.926,Z 399.592,A -85,B 0,C 180,E1 -6574.544,E2 -6574.544} C_VEL
LIN {X 0,Y 488.023,Z 395.609,A -85,B 0,C 180,E1 -6575.785,E2 -6575.785} C_VEL
LIN {X 0,Y 488.108,Z 392.397,A -85,B 0,C 180,E1 -6576.614,E2 -6576.614} C_VEL
LIN {X 0,Y 488.241,Z 386.376,A -85,B 0,C 180,E1 -6577.86,E2 -6577.86} C_VEL
LIN {X 0,Y 488.444,Z 380.28,A -85,B 0,C 180,E1 -6578.898,E2 -6578.898} C_VEL
LIN {X 0,Y 488.691,Z 374.58,A -85,B 0,C 180,E1 -6579.728,E2 -6579.728} C_VEL
LIN {X 0,Y 488.995,Z 366.024,A -85,B 0,C 180,E1 -6580.768,E2 -6580.768} C_VEL
LIN {X 0,Y 489.35,Z 357.843,A -85,B 0,C 180,E1 -6581.599,E2 -6581.599} C_VEL
LIN {X 0,Y 489.633,Z 349.328,A -85,B 0,C 180,E1 -6582.328,E2 -6582.328} C_VEL
LIN {X 0,Y 489.916,Z 341.099,A -85,B 0,C 180,E1 -6582.921,E2 -6582.921} C_VEL
LIN {X 0,Y 490.197,Z 331.854,A -85,B 0,C 180,E1 -6583.472,E2 -6583.472} C_VEL
LIN {X 0,Y 490.576,Z 322.054,A -85,B 0,C 180,E1 -6583.937,E2 -6583.937} C_VEL
LIN {X 0,Y 490.656,Z 316.9,A -85,B 0,C 180,E1 -6584.146,E2 -6584.146} C_VEL
LIN {X 0,Y 488.515,Z 303.537,A -85,B 0,C 180,E1 -6584.608,E2 -6584.608} C_VEL
LIN {X 0,Y 487.994,Z 300.235,A -85,B 0,C 180,E1 -6584.704,E2 -6584.704} C_VEL
LIN {X 0,Y 488.102,Z 293.2,A -85,B 0,C 180,E1 -6588.134,E2 -6588.134} C_VEL
LIN {X 0,Y 488.179,Z 287.303,A -85,B 0,C 180,E1 -6591.094,E2 -6591.094} C_VEL
LIN {X 0,Y 488.279,Z 282.135,A -85,B 0,C 180,E1 -6593.766,E2 -6593.766} C_VEL
LIN {X 0,Y 488.446,Z 276.341,A -85,B 0,C 180,E1 -6596.86,E2 -6596.86} C_VEL
LIN {X 0,Y 488.731,Z 270.293,A -85,B 0,C 180,E1 -6600.218,E2 -6600.218} C_VEL
LIN {X 0,Y 488.919,Z 265.368,A -85,B 0,C 180,E1 -6603.108,E2 -6603.108} C_VEL
LIN {X 0,Y 489.178,Z 259.999,A -85,B 0,C 180,E1 -6606.43,E2 -6606.43} C_VEL
LIN {X 0,Y 489.345,Z 255.811,A -85,B 0,C 180,E1 -6609.192,E2 -6609.192} C_VEL
LIN {X 0,Y 489.467,Z 252.242,A -85,B 0,C 180,E1 -6611.697,E2 -6611.697} C_VEL
LIN {X 0,Y 489.248,Z 249.072,A -85,B 0,C 180,E1 -6614.087,E2 -6614.087} C_VEL
LIN {X 0,Y 488.677,Z 245.116,A -85,B 0,C 180,E1 -6617.47,E2 -6617.47} C_VEL
LIN {X 0,Y 488.698,Z 245.112,A -85,B 0,C 180,E1 -6620.742,E2 -6620.742} C_VEL
LIN {X 0,Y 488.673,Z 245.116,A -85,B 0,C 180,E1 -6623.864,E2 -6623.864} C_VEL
LIN {X 0,Y 488.74,Z 245.101,A -85,B 0,C 180,E1 -6626.874,E2 -6626.874} C_VEL
LIN {X 0,Y 488.725,Z 245.108,A -85,B 0,C 180,E1 -6629.777,E2 -6629.777} C_VEL
LIN {X 0,Y 488.703,Z 245.105,A -85,B 0,C 180,E1 -6633.074,E2 -6633.074} C_VEL
LIN {X 0,Y 488.674,Z 245.112,A -85,B 0,C 180,E1 -6636.25,E2 -6636.25} C_VEL
LIN {X 0,Y 488.747,Z 245.101,A -85,B 0,C 180,E1 -6639.172,E2 -6639.172} C_VEL
LIN {X 0,Y 488.747,Z 245.108,A -85,B 0,C 180,E1 -6641.628,E2 -6641.628} C_VEL
LIN {X 0,Y 488.758,Z 245.1,A -85,B 0,C 180,E1 -6644.995,E2 -6644.995} C_VEL
LIN {X 0,Y 488.8,Z 245.093,A -85,B 0,C 180,E1 -6648.383,E2 -6648.383} C_VEL
LIN {X 0,Y 488.768,Z 245.102,A -85,B 0,C 180,E1 -6651.728,E2 -6651.728} C_VEL
LIN {X 0,Y 488.828,Z 245.09,A -85,B 0,C 180,E1 -6654.219,E2 -6654.219} C_VEL
LIN {X 0,Y 488.938,Z 245.081,A -85,B 0,C 180,E1 -6657.524,E2 -6657.524} C_VEL
LIN {X 0,Y 488.953,Z 245.075,A -85,B 0,C 180,E1 -6659.995,E2 -6659.995} C_VEL
LIN {X 0,Y 488.943,Z 245.076,A -85,B 0,C 180,E1 -6662.466,E2 -6662.466} C_VEL
LIN {X 0,Y 488.82,Z 245.092,A -85,B 0,C 180,E1 -6665.771,E2 -6665.771} C_VEL
LIN {X 0,Y 488.766,Z 245.098,A -85,B 0,C 180,E1 -6668.262,E2 -6668.262} C_VEL
LIN {X 0,Y 488.787,Z 245.096,A -85,B 0,C 180,E1 -6671.607,E2 -6671.607} C_VEL
LIN {X 0,Y 488.738,Z 245.108,A -85,B 0,C 180,E1 -6674.995,E2 -6674.995} C_VEL
LIN {X 0,Y 488.721,Z 245.107,A -85,B 0,C 180,E1 -6678.437,E2 -6678.437} C_VEL
LIN {X 0,Y 488.678,Z 245.112,A -85,B 0,C 180,E1 -6681.065,E2 -6681.065} C_VEL
LIN {X 0,Y 488.657,Z 245.111,A -85,B 0,C 180,E1 -6683.74,E2 -6683.74} C_VEL
LIN {X 0,Y 488.758,Z 245.102,A -85,B 0,C 180,E1 -6686.938,E2 -6686.938} C_VEL
LIN {X 0,Y 488.672,Z 245.116,A -85,B 0,C 180,E1 -6690.358,E2 -6690.358} C_VEL
LIN {X 0,Y 488.696,Z 245.106,A -85,B 0,C 180,E1 -6693.479,E2 -6693.479} C_VEL
LIN {X 0,Y 488.647,Z 245.121,A -85,B 0,C 180,E1 -6696.351,E2 -6696.351} C_VEL
LIN {X 0,Y 488.697,Z 245.106,A -85,B 0,C 180,E1 -6699.246,E2 -6699.246} C_VEL
LIN {X 0,Y 488.693,Z 245.11,A -85,B 0,C 180,E1 -6702.516,E2 -6702.516} C_VEL
LIN {X 0,Y 488.666,Z 245.11,A -85,B 0,C 180,E1 -6705.195,E2 -6705.195} C_VEL
LIN {X 0,Y 488.68,Z 245.112,A -85,B 0,C 180,E1 -6708.393,E2 -6708.393} C_VEL
LIN {X 0,Y 488.698,Z 245.106,A -85,B 0,C 180,E1 -6710.936,E2 -6710.936} C_VEL
LIN {X 0,Y 488.629,Z 245.123,A -85,B 0,C 180,E1 -6713.865,E2 -6713.865} C_VEL
LIN {X 0,Y 488.681,Z 245.108,A -85,B 0,C 180,E1 -6716.874,E2 -6716.874} C_VEL
LIN {X 0,Y 488.674,Z 245.117,A -85,B 0,C 180,E1 -6719.778,E2 -6719.778} C_VEL
LIN {X 0,Y 488.737,Z 245.102,A -85,B 0,C 180,E1 -6723.052,E2 -6723.052} C_VEL
LIN {X 0,Y 488.69,Z 245.107,A -85,B 0,C 180,E1 -6724.318,E2 -6724.318} C_VEL
LIN {X 0,Y 488.044,Z 245.19,A -85,B 0,C 180,E1 -6725.006,E2 -6725.006} C_VEL
LIN {X 0,Y 485.182,Z 245.551,A -85,B 0,C 180,E1 -6726.122,E2 -6726.122} C_VEL
LIN {X 0,Y 482.743,Z 245.856,A -85,B 0,C 180,E1 -6727.022,E2 -6727.022} C_VEL
LIN {X 0,Y 481.689,Z 245.985,A -85,B 0,C 180,E1 -6727.717,E2 -6727.717} C_VEL
LIN {X 0,Y 481.601,Z 245.993,A -85,B 0,C 180,E1 -6727.953,E2 -6727.953} C_VEL
LIN {X 0,Y 481.643,Z 245.985,A -85,B 0,C 180,E1 -6730.391,E2 -6730.391} C_VEL
LIN {X 0,Y 481.638,Z 245.991,A -85,B 0,C 180,E1 -6733.032,E2 -6733.032} C_VEL
LIN {X 0,Y 481.643,Z 245.991,A -85,B 0,C 180,E1 -6735.638,E2 -6735.638} C_VEL
LIN {X 0,Y 481.729,Z 245.976,A -85,B 0,C 180,E1 -6738.215,E2 -6738.215} C_VEL
LIN {X 0,Y 481.724,Z 245.98,A -85,B 0,C 180,E1 -6741.611,E2 -6741.611} C_VEL
LIN {X 0,Y 481.771,Z 245.972,A -85,B 0,C 180,E1 -6744.139,E2 -6744.139} C_VEL
LIN {X 0,Y 481.867,Z 245.962,A -85,B 0,C 180,E1 -6747.492,E2 -6747.492} C_VEL
LIN {X 0,Y 481.869,Z 245.96,A -85,B 0,C 180,E1 -6750,E2 -6750} C_VEL
LIN {X 0,Y 481.867,Z 245.962,A -85,B 0,C 180,E1 -6752.508,E2 -6752.508} C_VEL
LIN {X 0,Y 481.771,Z 245.972,A -85,B 0,C 180,E1 -6755.861,E2 -6755.861} C_VEL
LIN {X 0,Y 481.724,Z 245.98,A -85,B 0,C 180,E1 -6758.389,E2 -6758.389} C_VEL
LIN {X 0,Y 481.729,Z 245.976,A -85,B 0,C 180,E1 -6761.785,E2 -6761.785} C_VEL
LIN {X 0,Y 481.697,Z 245.982,A -85,B 0,C 180,E1 -6765.225,E2 -6765.225} C_VEL
LIN {X 0,Y 481.653,Z 245.989,A -85,B 0,C 180,E1 -6768.724,E2 -6768.724} C_VEL
LIN {X 0,Y 481.613,Z 245.989,A -85,B 0,C 180,E1 -6771.396,E2 -6771.396} C_VEL
LIN {X 0,Y 481.637,Z 245.99,A -85,B 0,C 180,E1 -6774.115,E2 -6774.115} C_VEL
LIN {X 0,Y 481.69,Z 245.979,A -85,B 0,C 180,E1 -6777.144,E2 -6777.144} C_VEL
LIN {X 0,Y 481.628,Z 245.989,A -85,B 0,C 180,E1 -6779.744,E2 -6779.744} C_VEL
LIN {X 0,Y 481.615,Z 245.991,A -85,B 0,C 180,E1 -6782.678,E2 -6782.678} C_VEL
LIN {X 0,Y 481.586,Z 245.995,A -85,B 0,C 180,E1 -6785.713,E2 -6785.713} C_VEL
LIN {X 0,Y 481.675,Z 245.982,A -85,B 0,C 180,E1 -6789.36,E2 -6789.36} C_VEL
LIN {X 0,Y 481.624,Z 245.993,A -85,B 0,C 180,E1 -6792.162,E2 -6792.162} C_VEL
LIN {X 0,Y 481.647,Z 245.99,A -85,B 0,C 180,E1 -6795.641,E2 -6795.641} C_VEL
LIN {X 0,Y 481.631,Z 245.991,A -85,B 0,C 180,E1 -6798.089,E2 -6798.089} C_VEL
LIN {X 0,Y 481.653,Z 245.985,A -85,B 0,C 180,E1 -6801.148,E2 -6801.148} C_VEL
LIN {X 0,Y 481.627,Z 245.987,A -85,B 0,C 180,E1 -6804.8,E2 -6804.8} C_VEL
LIN {X 0,Y 481.633,Z 245.991,A -85,B 0,C 180,E1 -6807.331,E2 -6807.331} C_VEL
LIN {X 0,Y 481.642,Z 245.985,A -85,B 0,C 180,E1 -6810.264,E2 -6810.264} C_VEL
LIN {X 0,Y 481.712,Z 245.98,A -85,B 0,C 180,E1 -6813.117,E2 -6813.117} C_VEL
LIN {X 0,Y 481.642,Z 245.987,A -85,B 0,C 180,E1 -6815.892,E2 -6815.892} C_VEL
LIN {X 0,Y 481.674,Z 245.986,A -85,B 0,C 180,E1 -6819.033,E2 -6819.033} C_VEL
LIN {X 0,Y 481.666,Z 245.982,A -85,B 0,C 180,E1 -6822.163,E2 -6822.163} C_VEL
LIN {X 0,Y 481.719,Z 245.979,A -85,B 0,C 180,E1 -6824.781,E2 -6824.781} C_VEL
LIN {X 0,Y 481.732,Z 245.974,A -85,B 0,C 180,E1 -6828.22,E2 -6828.22} C_VEL
LIN {X 0,Y 481.721,Z 245.976,A -85,B 0,C 180,E1 -6831.616,E2 -6831.616} C_VEL
LIN {X 0,Y 481.781,Z 245.968,A -85,B 0,C 180,E1 -6834.144,E2 -6834.144} C_VEL
LIN {X 0,Y 481.91,Z 245.952,A -85,B 0,C 180,E1 -6837.497,E2 -6837.497} C_VEL
LIN {X 0,Y 481.875,Z 245.963,A -85,B 0,C 180,E1 -6840.84,E2 -6840.84} C_VEL
LIN {X 0,Y 481.904,Z 245.958,A -85,B 0,C 180,E1 -6842.512,E2 -6842.512} C_VEL
LIN {X 0,Y 481.789,Z 245.967,A -85,B 0,C 180,E1 -6845.865,E2 -6845.865} C_VEL
LIN {X 0,Y 481.723,Z 245.981,A -85,B 0,C 180,E1 -6848.393,E2 -6848.393} C_VEL
LIN {X 0,Y 481.746,Z 245.973,A -85,B 0,C 180,E1 -6851.789,E2 -6851.789} C_VEL
LIN {X 0,Y 481.74,Z 245.973,A -85,B 0,C 180,E1 -6855.228,E2 -6855.228} C_VEL
LIN {X 0,Y 481.707,Z 245.98,A -85,B 0,C 180,E1 -6858.726,E2 -6858.726} C_VEL
LIN {X 0,Y 481.646,Z 245.985,A -85,B 0,C 180,E1 -6861.399,E2 -6861.399} C_VEL
LIN {X 0,Y 481.653,Z 245.991,A -85,B 0,C 180,E1 -6864.118,E2 -6864.118} C_VEL
LIN {X 0,Y 481.677,Z 245.981,A -85,B 0,C 180,E1 -6867.125,E2 -6867.125} C_VEL
LIN {X 0,Y 481.673,Z 245.986,A -85,B 0,C 180,E1 -6869.745,E2 -6869.745} C_VEL
LIN {X 0,Y 481.675,Z 245.981,A -85,B 0,C 180,E1 -6872.677,E2 -6872.677} C_VEL
LIN {X 0,Y 481.635,Z 245.992,A -85,B 0,C 180,E1 -6875.713,E2 -6875.713} C_VEL
LIN {X 0,Y 481.67,Z 245.986,A -85,B 0,C 180,E1 -6878.863,E2 -6878.863} C_VEL
LIN {X 0,Y 481.638,Z 245.993,A -85,B 0,C 180,E1 -6882.165,E2 -6882.165} C_VEL
LIN {X 0,Y 482,Z 248.426,A -85,B 0,C 180,E1 -6884.421,E2 -6884.421} C_VEL
LIN {X 0,Y 482.349,Z 251.35,A -85,B 0,C 180,E1 -6886.781,E2 -6886.781} C_VEL
LIN {X 0,Y 482.38,Z 254.673,A -85,B 0,C 180,E1 -6889.257,E2 -6889.257} C_VEL
LIN {X 0,Y 482.207,Z 259.017,A -85,B 0,C 180,E1 -6892.257,E2 -6892.257} C_VEL
LIN {X 0,Y 481.993,Z 263.786,A -85,B 0,C 180,E1 -6895.344,E2 -6895.344} C_VEL
LIN {X 0,Y 481.756,Z 268.661,A -85,B 0,C 180,E1 -6898.321,E2 -6898.321} C_VEL
LIN {X 0,Y 481.529,Z 273.631,A -85,B 0,C 180,E1 -6901.208,E2 -6901.208} C_VEL
LIN {X 0,Y 481.321,Z 278.668,A -85,B 0,C 180,E1 -6904.022,E2 -6904.022} C_VEL
LIN {X 0,Y 481.188,Z 284.11,A -85,B 0,C 180,E1 -6906.952,E2 -6906.952} C_VEL
LIN {X 0,Y 481.097,Z 288.942,A -85,B 0,C 180,E1 -6909.477,E2 -6909.477} C_VEL
LIN {X 0,Y 481.003,Z 294.146,A -85,B 0,C 180,E1 -6912.132,E2 -6912.132} C_VEL
LIN {X 0,Y 480.941,Z 300.155,A -85,B 0,C 180,E1 -6915.092,E2 -6915.092} C_VEL
LIN {X 0,Y 482.626,Z 310.581,A -85,B 0,C 180,E1 -6915.412,E2 -6915.412} C_VEL
LIN {X 0,Y 483.779,Z 319.283,A -85,B 0,C 180,E1 -6915.756,E2 -6915.756} C_VEL
LIN {X 0,Y 483.477,Z 328.64,A -85,B 0,C 180,E1 -6916.176,E2 -6916.176} C_VEL
LIN {X 0,Y 483.067,Z 338.785,A -85,B 0,C 180,E1 -6916.754,E2 -6916.754} C_VEL
LIN {X 0,Y 482.673,Z 347.779,A -85,B 0,C 180,E1 -6917.385,E2 -6917.385} C_VEL
LIN {X 0,Y 482.408,Z 356.572,A -85,B 0,C 180,E1 -6918.131,E2 -6918.131} C_VEL
LIN {X 0,Y 482.121,Z 363.91,A -85,B 0,C 180,E1 -6918.864,E2 -6918.864} C_VEL
LIN {X 0,Y 481.757,Z 371.129,A -85,B 0,C 180,E1 -6919.706,E2 -6919.706} C_VEL
LIN {X 0,Y 481.513,Z 377.332,A -85,B 0,C 180,E1 -6920.549,E2 -6920.549} C_VEL
LIN {X 0,Y 481.275,Z 383.87,A -85,B 0,C 180,E1 -6921.603,E2 -6921.603} C_VEL
LIN {X 0,Y 481.121,Z 388.371,A -85,B 0,C 180,E1 -6922.446,E2 -6922.446} C_VEL
LIN {X 0,Y 480.93,Z 394.308,A -85,B 0,C 180,E1 -6923.83,E2 -6923.83} C_VEL
LIN {X 0,Y 480.903,Z 398.182,A -85,B 0,C 180,E1 -6924.97,E2 -6924.97} C_VEL
LIN {X 0,Y 480.832,Z 400.545,A -85,B 0,C 180,E1 -6925.809,E2 -6925.809} C_VEL
LIN {X 0,Y 480.874,Z 402.343,A -85,B 0,C 180,E1 -6926.649,E2 -6926.649} C_VEL
LIN {X 0,Y 480.796,Z 404.782,A -85,B 0,C 180,E1 -6928.325,E2 -6928.325} C_VEL
LIN {X 0,Y 480.763,Z 405.368,A -85,B 0,C 180,E1 -6929.162,E2 -6929.162} C_VEL
LIN {X 0,Y 480.763,Z 405.368,A -85,B 0,C 180,E1 -6930.838,E2 -6930.838} C_VEL
LIN {X 0,Y 480.796,Z 404.782,A -85,B 0,C 180,E1 -6931.675,E2 -6931.675} C_VEL
LIN {X 0,Y 480.874,Z 402.343,A -85,B 0,C 180,E1 -6933.351,E2 -6933.351} C_VEL
LIN {X 0,Y 480.845,Z 399.397,A -85,B 0,C 180,E1 -6934.611,E2 -6934.611} C_VEL
LIN {X 0,Y 480.928,Z 395.413,A -85,B 0,C 180,E1 -6935.871,E2 -6935.871} C_VEL
LIN {X 0,Y 481.024,Z 392.201,A -85,B 0,C 180,E1 -6936.712,E2 -6936.712} C_VEL
LIN {X 0,Y 481.186,Z 386.181,A -85,B 0,C 180,E1 -6937.975,E2 -6937.975} C_VEL
LIN {X 0,Y 481.407,Z 380.085,A -85,B 0,C 180,E1 -6939.029,E2 -6939.029} C_VEL
LIN {X 0,Y 481.664,Z 374.385,A -85,B 0,C 180,E1 -6939.872,E2 -6939.872} C_VEL
LIN {X 0,Y 482.013,Z 365.829,A -85,B 0,C 180,E1 -6940.926,E2 -6940.926} C_VEL
LIN {X 0,Y 482.377,Z 357.648,A -85,B 0,C 180,E1 -6941.769,E2 -6941.769} C_VEL
LIN {X 0,Y 482.668,Z 349.243,A -85,B 0,C 180,E1 -6942.5,E2 -6942.5} C_VEL
LIN {X 0,Y 482.989,Z 340.904,A -85,B 0,C 180,E1 -6943.109,E2 -6943.109} C_VEL
LIN {X 0,Y 483.356,Z 330.653,A -85,B 0,C 180,E1 -6943.72,E2 -6943.72} C_VEL
LIN {X 0,Y 483.735,Z 320.571,A -85,B 0,C 180,E1 -6944.192,E2 -6944.192} C_VEL
LIN {X 0,Y 483.566,Z 316.699,A -85,B 0,C 180,E1 -6944.358,E2 -6944.358} C_VEL
LIN {X 0,Y 481.311,Z 302.666,A -85,B 0,C 180,E1 -6944.845,E2 -6944.845} C_VEL
LIN {X 0,Y 480.928,Z 300.077,A -85,B 0,C 180,E1 -6944.925,E2 -6944.925} C_VEL
LIN {X 0,Y 481.019,Z 293.391,A -85,B 0,C 180,E1 -6948.247,E2 -6948.247} C_VEL
LIN {X 0,Y 481.104,Z 287.206,A -85,B 0,C 180,E1 -6951.419,E2 -6951.419} C_VEL
LIN {X 0,Y 481.239,Z 282.065,A -85,B 0,C 180,E1 -6954.136,E2 -6954.136} C_VEL
LIN {X 0,Y 481.398,Z 276.712,A -85,B 0,C 180,E1 -6957.054,E2 -6957.054} C_VEL
LIN {X 0,Y 481.606,Z 271.941,A -85,B 0,C 180,E1 -6959.745,E2 -6959.745} C_VEL
LIN {X 0,Y 481.848,Z 267.008,A -85,B 0,C 180,E1 -6962.66,E2 -6962.66} C_VEL
LIN {X 0,Y 482.061,Z 262.172,A -85,B 0,C 180,E1 -6965.672,E2 -6965.672} C_VEL
LIN {X 0,Y 482.279,Z 257.43,A -85,B 0,C 180,E1 -6968.8,E2 -6968.8} C_VEL
LIN {X 0,Y 482.412,Z 254.362,A -85,B 0,C 180,E1 -6970.962,E2 -6970.962} C_VEL
LIN {X 0,Y 482.346,Z 251.312,A -85,B 0,C 180,E1 -6973.234,E2 -6973.234} C_VEL
LIN {X 0,Y 481.964,Z 248.389,A -85,B 0,C 180,E1 -6975.602,E2 -6975.602} C_VEL
LIN {X 0,Y 481.638,Z 245.992,A -85,B 0,C 180,E1 -6977.835,E2 -6977.835} C_VEL
LIN {X 0,Y 481.67,Z 245.986,A -85,B 0,C 180,E1 -6981.137,E2 -6981.137} C_VEL
LIN {X 0,Y 481.662,Z 245.987,A -85,B 0,C 180,E1 -6984.794,E2 -6984.794} C_VEL
LIN {X 0,Y 481.66,Z 245.988,A -85,B 0,C 180,E1 -6987.808,E2 -6987.808} C_VEL
LIN {X 0,Y 481.647,Z 245.984,A -85,B 0,C 180,E1 -6991.101,E2 -6991.101} C_VEL
LIN {X 0,Y 481.651,Z 245.99,A -85,B 0,C 180,E1 -6994.036,E2 -6994.036} C_VEL
LIN {X 0,Y 481.676,Z 245.981,A -85,B 0,C 180,E1 -6996.808,E2 -6996.808} C_VEL
LIN {X 0,Y 481.695,Z 245.983,A -85,B 0,C 180,E1 -6999.499,E2 -6999.499} C_VEL
LIN {X 0,Y 481.686,Z 245.982,A -85,B 0,C 180,E1 -7002.154,E2 -7002.154} C_VEL
LIN {X 0,Y 481.74,Z 245.973,A -85,B 0,C 180,E1 -7004.772,E2 -7004.772} C_VEL
LIN {X 0,Y 481.746,Z 245.973,A -85,B 0,C 180,E1 -7008.211,E2 -7008.211} C_VEL
LIN {X 0,Y 481.723,Z 245.981,A -85,B 0,C 180,E1 -7011.607,E2 -7011.607} C_VEL
LIN {X 0,Y 481.789,Z 245.967,A -85,B 0,C 180,E1 -7014.135,E2 -7014.135} C_VEL
LIN {X 0,Y 481.904,Z 245.958,A -85,B 0,C 180,E1 -7017.488,E2 -7017.488} C_VEL
LIN {X 0,Y 481.924,Z 245.95,A -85,B 0,C 180,E1 -7019.995,E2 -7019.995} C_VEL
LIN {X 0,Y 481.91,Z 245.952,A -85,B 0,C 180,E1 -7022.503,E2 -7022.503} C_VEL
LIN {X 0,Y 481.781,Z 245.968,A -85,B 0,C 180,E1 -7025.856,E2 -7025.856} C_VEL
LIN {X 0,Y 481.721,Z 245.976,A -85,B 0,C 180,E1 -7028.384,E2 -7028.384} C_VEL
LIN {X 0,Y 481.732,Z 245.974,A -85,B 0,C 180,E1 -7031.78,E2 -7031.78} C_VEL
LIN {X 0,Y 481.719,Z 245.979,A -85,B 0,C 180,E1 -7035.219,E2 -7035.219} C_VEL
LIN {X 0,Y 481.682,Z 245.988,A -85,B 0,C 180,E1 -7038.717,E2 -7038.717} C_VEL
LIN {X 0,Y 481.617,Z 245.989,A -85,B 0,C 180,E1 -7041.389,E2 -7041.389} C_VEL
LIN {X 0,Y 481.642,Z 245.987,A -85,B 0,C 180,E1 -7044.108,E2 -7044.108} C_VEL
LIN {X 0,Y 481.713,Z 245.978,A -85,B 0,C 180,E1 -7047.134,E2 -7047.134} C_VEL
LIN {X 0,Y 481.642,Z 245.985,A -85,B 0,C 180,E1 -7049.736,E2 -7049.736} C_VEL
LIN {X 0,Y 481.633,Z 245.991,A -85,B 0,C 180,E1 -7052.669,E2 -7052.669} C_VEL
LIN {X 0,Y 481.602,Z 245.991,A -85,B 0,C 180,E1 -7055.704,E2 -7055.704} C_VEL
LIN {X 0,Y 481.669,Z 245.982,A -85,B 0,C 180,E1 -7059.349,E2 -7059.349} C_VEL
LIN {X 0,Y 481.632,Z 245.994,A -85,B 0,C 180,E1 -7062.153,E2 -7062.153} C_VEL
LIN {X 0,Y 481.645,Z 245.989,A -85,B 0,C 180,E1 -7064.449,E2 -7064.449} C_VEL
LIN {X 0,Y 481.624,Z 245.993,A -85,B 0,C 180,E1 -7067.838,E2 -7067.838} C_VEL
LIN {X 0,Y 481.653,Z 245.984,A -85,B 0,C 180,E1 -7071.14,E2 -7071.14} C_VEL
LIN {X 0,Y 481.611,Z 245.989,A -85,B 0,C 180,E1 -7074.791,E2 -7074.791} C_VEL
LIN {X 0,Y 481.615,Z 245.991,A -85,B 0,C 180,E1 -7077.322,E2 -7077.322} C_VEL
LIN {X 0,Y 481.628,Z 245.989,A -85,B 0,C 180,E1 -7080.256,E2 -7080.256} C_VEL
LIN {X 0,Y 481.691,Z 245.98,A -85,B 0,C 180,E1 -7083.109,E2 -7083.109} C_VEL
LIN {X 0,Y 481.637,Z 245.99,A -85,B 0,C 180,E1 -7085.885,E2 -7085.885} C_VEL
LIN {X 0,Y 481.601,Z 245.993,A -85,B 0,C 180,E1 -7087.953,E2 -7087.953} C_VEL
LIN {X 0,Y 480.931,Z 246.074,A -85,B 0,C 180,E1 -7088.651,E2 -7088.651} C_VEL
LIN {X 0,Y 478.093,Z 246.434,A -85,B 0,C 180,E1 -7089.785,E2 -7089.785} C_VEL
LIN {X 0,Y 475.702,Z 246.732,A -85,B 0,C 180,E1 -7090.699,E2 -7090.699} C_VEL
LIN {X 0,Y 474.682,Z 246.86,A -85,B 0,C 180,E1 -7091.405,E2 -7091.405} C_VEL
LIN {X 0,Y 474.602,Z 246.867,A -85,B 0,C 180,E1 -7091.644,E2 -7091.644} C_VEL
LIN {X 0,Y 474.651,Z 246.859,A -85,B 0,C 180,E1 -7094.543,E2 -7094.543} C_VEL
LIN {X 0,Y 474.672,Z 246.856,A -85,B 0,C 180,E1 -7098.037,E2 -7098.037} C_VEL
LIN {X 0,Y 474.682,Z 246.858,A -85,B 0,C 180,E1 -7101.486,E2 -7101.486} C_VEL
LIN {X 0,Y 474.733,Z 246.849,A -85,B 0,C 180,E1 -7104.052,E2 -7104.052} C_VEL
LIN {X 0,Y 474.834,Z 246.839,A -85,B 0,C 180,E1 -7107.455,E2 -7107.455} C_VEL
LIN {X 0,Y 474.841,Z 246.836,A -85,B 0,C 180,E1 -7110,E2 -7110} C_VEL
LIN {X 0,Y 474.834,Z 246.839,A -85,B 0,C 180,E1 -7112.545,E2 -7112.545} C_VEL
LIN {X 0,Y 474.733,Z 246.849,A -85,B 0,C 180,E1 -7115.948,E2 -7115.948} C_VEL
LIN {X 0,Y 474.682,Z 246.858,A -85,B 0,C 180,E1 -7118.514,E2 -7118.514} C_VEL
LIN {X 0,Y 474.672,Z 246.856,A -85,B 0,C 180,E1 -7121.963,E2 -7121.963} C_VEL
LIN {X 0,Y 474.648,Z 246.859,A -85,B 0,C 180,E1 -7125.784,E2 -7125.784} C_VEL
LIN {X 0,Y 474.603,Z 246.864,A -85,B 0,C 180,E1 -7129.012,E2 -7129.012} C_VEL
LIN {X 0,Y 474.581,Z 246.865,A -85,B 0,C 180,E1 -7131.729,E2 -7131.729} C_VEL
LIN {X 0,Y 474.615,Z 246.867,A -85,B 0,C 180,E1 -7134.495,E2 -7134.495} C_VEL
LIN {X 0,Y 474.638,Z 246.857,A -85,B 0,C 180,E1 -7137.342,E2 -7137.342} C_VEL
LIN {X 0,Y 474.55,Z 246.87,A -85,B 0,C 180,E1 -7140.815,E2 -7140.815} C_VEL
LIN {X 0,Y 474.581,Z 246.87,A -85,B 0,C 180,E1 -7143.988,E2 -7143.988} C_VEL
LIN {X 0,Y 474.521,Z 246.872,A -85,B 0,C 180,E1 -7146.904,E2 -7146.904} C_VEL
LIN {X 0,Y 474.618,Z 246.863,A -85,B 0,C 180,E1 -7149.658,E2 -7149.658} C_VEL
LIN {X 0,Y 474.601,Z 246.862,A -85,B 0,C 180,E1 -7152.934,E2 -7152.934} C_VEL
LIN {X 0,Y 474.616,Z 246.868,A -85,B 0,C 180,E1 -7155.906,E2 -7155.906} C_VEL
LIN {X 0,Y 474.601,Z 246.863,A -85,B 0,C 180,E1 -7159.043,E2 -7159.043} C_VEL
LIN {X 0,Y 474.573,Z 246.874,A -85,B 0,C 180,E1 -7161.708,E2 -7161.708} C_VEL
LIN {X 0,Y 474.589,Z 246.864,A -85,B 0,C 180,E1 -7164.731,E2 -7164.731} C_VEL
LIN {X 0,Y 474.597,Z 246.868,A -85,B 0,C 180,E1 -7167.793,E2 -7167.793} C_VEL
LIN {X 0,Y 474.588,Z 246.865,A -85,B 0,C 180,E1 -7170.89,E2 -7170.89} C_VEL
LIN {X 0,Y 474.626,Z 246.864,A -85,B 0,C 180,E1 -7173.634,E2 -7173.634} C_VEL
LIN {X 0,Y 474.605,Z 246.862,A -85,B 0,C 180,E1 -7176.647,E2 -7176.647} C_VEL
LIN {X 0,Y 474.627,Z 246.859,A -85,B 0,C 180,E1 -7180.095,E2 -7180.095} C_VEL
LIN {X 0,Y 474.613,Z 246.863,A -85,B 0,C 180,E1 -7182.779,E2 -7182.779} C_VEL
LIN {X 0,Y 474.624,Z 246.863,A -85,B 0,C 180,E1 -7185.426,E2 -7185.426} C_VEL
LIN {X 0,Y 474.685,Z 246.852,A -85,B 0,C 180,E1 -7188.043,E2 -7188.043} C_VEL
LIN {X 0,Y 474.693,Z 246.853,A -85,B 0,C 180,E1 -7191.491,E2 -7191.491} C_VEL
LIN {X 0,Y 474.744,Z 246.844,A -85,B 0,C 180,E1 -7194.057,E2 -7194.057} C_VEL
LIN {X 0,Y 474.877,Z 246.829,A -85,B 0,C 180,E1 -7197.46,E2 -7197.46} C_VEL
LIN {X 0,Y 474.895,Z 246.826,A -85,B 0,C 180,E1 -7200.005,E2 -7200.005} C_VEL
LIN {X 0,Y 474.87,Z 246.835,A -85,B 0,C 180,E1 -7202.55,E2 -7202.55} C_VEL
LIN {X 0,Y 474.752,Z 246.844,A -85,B 0,C 180,E1 -7205.953,E2 -7205.953} C_VEL
LIN {X 0,Y 474.696,Z 246.858,A -85,B 0,C 180,E1 -7208.519,E2 -7208.519} C_VEL
LIN {X 0,Y 474.7,Z 246.852,A -85,B 0,C 180,E1 -7211.967,E2 -7211.967} C_VEL
LIN {X 0,Y 474.697,Z 246.85,A -85,B 0,C 180,E1 -7215.46,E2 -7215.46} C_VEL
LIN {X 0,Y 474.661,Z 246.855,A -85,B 0,C 180,E1 -7219.014,E2 -7219.014} C_VEL
LIN {X 0,Y 474.589,Z 246.866,A -85,B 0,C 180,E1 -7221.733,E2 -7221.733} C_VEL
LIN {X 0,Y 474.631,Z 246.862,A -85,B 0,C 180,E1 -7224.498,E2 -7224.498} C_VEL
LIN {X 0,Y 474.64,Z 246.858,A -85,B 0,C 180,E1 -7227.327,E2 -7227.327} C_VEL
LIN {X 0,Y 474.604,Z 246.867,A -85,B 0,C 180,E1 -7230.234,E2 -7230.234} C_VEL
LIN {X 0,Y 474.63,Z 246.859,A -85,B 0,C 180,E1 -7233.225,E2 -7233.225} C_VEL
LIN {X 0,Y 474.588,Z 246.869,A -85,B 0,C 180,E1 -7236.327,E2 -7236.327} C_VEL
LIN {X 0,Y 474.627,Z 246.867,A -85,B 0,C 180,E1 -7239.551,E2 -7239.551} C_VEL
LIN {X 0,Y 474.621,Z 247.095,A -85,B 0,C 180,E1 -7242.238,E2 -7242.238} C_VEL
LIN {X 0,Y 475.118,Z 250.567,A -85,B 0,C 180,E1 -7245.24,E2 -7245.24} C_VEL
LIN {X 0,Y 475.386,Z 253.63,A -85,B 0,C 180,E1 -7247.666,E2 -7247.666} C_VEL
LIN {X 0,Y 475.302,Z 257.517,A -85,B 0,C 180,E1 -7250.521,E2 -7250.521} C_VEL
LIN {X 0,Y 475.088,Z 262.237,A -85,B 0,C 180,E1 -7253.722,E2 -7253.722} C_VEL
LIN {X 0,Y 474.841,Z 267.036,A -85,B 0,C 180,E1 -7256.797,E2 -7256.797} C_VEL
LIN {X 0,Y 474.574,Z 271.956,A -85,B 0,C 180,E1 -7259.768,E2 -7259.768} C_VEL
LIN {X 0,Y 474.364,Z 277.086,A -85,B 0,C 180,E1 -7262.744,E2 -7262.744} C_VEL
LIN {X 0,Y 474.172,Z 281.994,A -85,B 0,C 180,E1 -7265.481,E2 -7265.481} C_VEL
LIN {X 0,Y 474.031,Z 287.125,A -85,B 0,C 180,E1 -7268.245,E2 -7268.245} C_VEL
LIN {X 0,Y 473.93,Z 293.598,A -85,B 0,C 180,E1 -7271.64,E2 -7271.64} C_VEL
LIN {X 0,Y 473.833,Z 300.026,A -85,B 0,C 180,E1 -7274.865,E2 -7274.865} C_VEL
LIN {X 0,Y 475.579,Z 310.643,A -85,B 0,C 180,E1 -7275.199,E2 -7275.199} C_VEL
LIN {X 0,Y 476.849,Z 319.087,A -85,B 0,C 180,E1 -7275.545,E2 -7275.545} C_VEL
LIN {X 0,Y 476.576,Z 328.445,A -85,B 0,C 180,E1 -7275.972,E2 -7275.972} C_VEL
LIN {X 0,Y 476.113,Z 338.912,A -85,B 0,C 180,E1 -7276.578,E2 -7276.578} C_VEL
LIN {X 0,Y 475.727,Z 347.584,A -85,B 0,C 180,E1 -7277.197,E2 -7277.197} C_VEL
LIN {X 0,Y 475.45,Z 355.471,A -85,B 0,C 180,E1 -7277.868,E2 -7277.868} C_VEL
LIN {X 0,Y 475.135,Z 363.715,A -85,B 0,C 180,E1 -7278.698,E2 -7278.698} C_VEL
LIN {X 0,Y 474.747,Z 370.934,A -85,B 0,C 180,E1 -7279.552,E2 -7279.552} C_VEL
LIN {X 0,Y 474.488,Z 377.137,A -85,B 0,C 180,E1 -7280.408,E2 -7280.408} C_VEL
LIN {X 0,Y 474.206,Z 383.674,A -85,B 0,C 180,E1 -7281.477,E2 -7281.477} C_VEL
LIN {X 0,Y 474.047,Z 388.175,A -85,B 0,C 180,E1 -7282.332,E2 -7282.332} C_VEL
LIN {X 0,Y 473.879,Z 393.466,A -85,B 0,C 180,E1 -7283.559,E2 -7283.559} C_VEL
LIN {X 0,Y 473.833,Z 397.988,A -85,B 0,C 180,E1 -7284.894,E2 -7284.894} C_VEL
LIN {X 0,Y 473.739,Z 400.35,A -85,B 0,C 180,E1 -7285.746,E2 -7285.746} C_VEL
LIN {X 0,Y 473.769,Z 402.148,A -85,B 0,C 180,E1 -7286.598,E2 -7286.598} C_VEL
LIN {X 0,Y 473.701,Z 404.587,A -85,B 0,C 180,E1 -7288.3,E2 -7288.3} C_VEL
LIN {X 0,Y 473.691,Z 405.174,A -85,B 0,C 180,E1 -7289.15,E2 -7289.15} C_VEL
LIN {X 0,Y 473.691,Z 405.174,A -85,B 0,C 180,E1 -7290.85,E2 -7290.85} C_VEL
LIN {X 0,Y 473.701,Z 404.587,A -85,B 0,C 180,E1 -7291.7,E2 -7291.7} C_VEL
LIN {X 0,Y 473.769,Z 402.148,A -85,B 0,C 180,E1 -7293.402,E2 -7293.402} C_VEL
LIN {X 0,Y 473.768,Z 399.202,A -85,B 0,C 180,E1 -7294.68,E2 -7294.68} C_VEL
LIN {X 0,Y 473.836,Z 395.218,A -85,B 0,C 180,E1 -7295.959,E2 -7295.959} C_VEL
LIN {X 0,Y 474.015,Z 390.092,A -85,B 0,C 180,E1 -7297.24,E2 -7297.24} C_VEL
LIN {X 0,Y 474.171,Z 384.83,A -85,B 0,C 180,E1 -7298.309,E2 -7298.309} C_VEL
LIN {X 0,Y 474.42,Z 378.513,A -85,B 0,C 180,E1 -7299.378,E2 -7299.378} C_VEL
LIN {X 0,Y 474.657,Z 372.561,A -85,B 0,C 180,E1 -7300.234,E2 -7300.234} C_VEL
LIN {X 0,Y 475.005,Z 365.634,A -85,B 0,C 180,E1 -7301.089,E2 -7301.089} C_VEL
LIN {X 0,Y 475.402,Z 357.453,A -85,B 0,C 180,E1 -7301.944,E2 -7301.944} C_VEL
LIN {X 0,Y 475.671,Z 349.046,A -85,B 0,C 180,E1 -7302.687,E2 -7302.687} C_VEL
LIN {X 0,Y 476.062,Z 340.709,A -85,B 0,C 180,E1 -7303.303,E2 -7303.303} C_VEL
LIN {X 0,Y 476.427,Z 330.457,A -85,B 0,C 180,E1 -7303.924,E2 -7303.924} C_VEL
LIN {X 0,Y 476.805,Z 321.664,A -85,B 0,C 180,E1 -7304.348,E2 -7304.348} C_VEL
LIN {X 0,Y 476.513,Z 316.602,A -85,B 0,C 180,E1 -7304.571,E2 -7304.571} C_VEL
LIN {X 0,Y 474.239,Z 302.347,A -85,B 0,C 180,E1 -7305.074,E2 -7305.074} C_VEL
LIN {X 0,Y 473.837,Z 299.904,A -85,B 0,C 180,E1 -7305.16,E2 -7305.16} C_VEL
LIN {X 0,Y 473.93,Z 293.587,A -85,B 0,C 180,E1 -7308.36,E2 -7308.36} C_VEL
LIN {X 0,Y 474.03,Z 287.109,A -85,B 0,C 180,E1 -7311.755,E2 -7311.755} C_VEL
LIN {X 0,Y 474.173,Z 281.993,A -85,B 0,C 180,E1 -7314.519,E2 -7314.519} C_VEL
LIN {X 0,Y 474.365,Z 276.924,A -85,B 0,C 180,E1 -7317.34,E2 -7317.34} C_VEL
LIN {X 0,Y 474.574,Z 271.916,A -85,B 0,C 180,E1 -7320.232,E2 -7320.232} C_VEL
LIN {X 0,Y 474.84,Z 267.03,A -85,B 0,C 180,E1 -7323.204,E2 -7323.204} C_VEL
LIN {X 0,Y 475.087,Z 262.2,A -85,B 0,C 180,E1 -7326.278,E2 -7326.278} C_VEL
LIN {X 0,Y 475.303,Z 257.513,A -85,B 0,C 180,E1 -7329.479,E2 -7329.479} C_VEL
LIN {X 0,Y 475.411,Z 254.448,A -85,B 0,C 180,E1 -7331.699,E2 -7331.699} C_VEL
LIN {X 0,Y 475.242,Z 251.448,A -85,B 0,C 180,E1 -7334.03,E2 -7334.03} C_VEL
LIN {X 0,Y 474.729,Z 247.868,A -85,B 0,C 180,E1 -7337.075,E2 -7337.075} C_VEL
LIN {X 0,Y 474.612,Z 246.869,A -85,B 0,C 180,E1 -7338.21,E2 -7338.21} C_VEL
LIN {X 0,Y 474.613,Z 246.866,A -85,B 0,C 180,E1 -7341.539,E2 -7341.539} C_VEL
LIN {X 0,Y 474.624,Z 246.864,A -85,B 0,C 180,E1 -7344.722,E2 -7344.722} C_VEL
LIN {X 0,Y 474.639,Z 246.862,A -85,B 0,C 180,E1 -7347.784,E2 -7347.784} C_VEL
LIN {X 0,Y 474.604,Z 246.862,A -85,B 0,C 180,E1 -7350.886,E2 -7350.886} C_VEL
LIN {X 0,Y 474.597,Z 246.867,A -85,B 0,C 180,E1 -7353.621,E2 -7353.621} C_VEL
LIN {X 0,Y 474.636,Z 246.858,A -85,B 0,C 180,E1 -7356.638,E2 -7356.638} C_VEL
LIN {X 0,Y 474.652,Z 246.859,A -85,B 0,C 180,E1 -7360.085,E2 -7360.085} C_VEL
LIN {X 0,Y 474.632,Z 246.858,A -85,B 0,C 180,E1 -7362.77,E2 -7362.77} C_VEL
LIN {X 0,Y 474.643,Z 246.863,A -85,B 0,C 180,E1 -7365.417,E2 -7365.417} C_VEL
LIN {X 0,Y 474.7,Z 246.852,A -85,B 0,C 180,E1 -7368.033,E2 -7368.033} C_VEL
LIN {X 0,Y 474.696,Z 246.858,A -85,B 0,C 180,E1 -7371.481,E2 -7371.481} C_VEL
LIN {X 0,Y 474.752,Z 246.844,A -85,B 0,C 180,E1 -7374.047,E2 -7374.047} C_VEL
LIN {X 0,Y 474.87,Z 246.835,A -85,B 0,C 180,E1 -7377.45,E2 -7377.45} C_VEL
LIN {X 0,Y 474.895,Z 246.826,A -85,B 0,C 180,E1 -7379.995,E2 -7379.995} C_VEL
LIN {X 0,Y 474.877,Z 246.829,A -85,B 0,C 180,E1 -7382.54,E2 -7382.54} C_VEL
LIN {X 0,Y 474.744,Z 246.844,A -85,B 0,C 180,E1 -7385.943,E2 -7385.943} C_VEL
LIN {X 0,Y 474.693,Z 246.853,A -85,B 0,C 180,E1 -7388.509,E2 -7388.509} C_VEL
LIN {X 0,Y 474.685,Z 246.852,A -85,B 0,C 180,E1 -7391.957,E2 -7391.957} C_VEL
LIN {X 0,Y 474.676,Z 246.854,A -85,B 0,C 180,E1 -7395.45,E2 -7395.45} C_VEL
LIN {X 0,Y 474.636,Z 246.863,A -85,B 0,C 180,E1 -7399.005,E2 -7399.005} C_VEL
LIN {X 0,Y 474.559,Z 246.867,A -85,B 0,C 180,E1 -7401.724,E2 -7401.724} C_VEL
LIN {X 0,Y 474.623,Z 246.866,A -85,B 0,C 180,E1 -7404.488,E2 -7404.488} C_VEL
LIN {X 0,Y 474.648,Z 246.857,A -85,B 0,C 180,E1 -7407.329,E2 -7407.329} C_VEL
LIN {X 0,Y 474.567,Z 246.87,A -85,B 0,C 180,E1 -7410.805,E2 -7410.805} C_VEL
LIN {X 0,Y 474.599,Z 246.865,A -85,B 0,C 180,E1 -7413.979,E2 -7413.979} C_VEL
LIN {X 0,Y 474.532,Z 246.872,A -85,B 0,C 180,E1 -7416.895,E2 -7416.895} C_VEL
LIN {X 0,Y 474.605,Z 246.863,A -85,B 0,C 180,E1 -7419.646,E2 -7419.646} C_VEL
LIN {X 0,Y 474.615,Z 246.861,A -85,B 0,C 180,E1 -7422.924,E2 -7422.924} C_VEL
LIN {X 0,Y 474.569,Z 246.871,A -85,B 0,C 180,E1 -7425.892,E2 -7425.892} C_VEL
LIN {X 0,Y 474.595,Z 246.863,A -85,B 0,C 180,E1 -7429.034,E2 -7429.034} C_VEL
LIN {X 0,Y 474.567,Z 246.871,A -85,B 0,C 180,E1 -7431.698,E2 -7431.698} C_VEL
LIN {X 0,Y 474.573,Z 246.866,A -85,B 0,C 180,E1 -7434.722,E2 -7434.722} C_VEL
LIN {X 0,Y 474.579,Z 246.873,A -85,B 0,C 180,E1 -7437.784,E2 -7437.784} C_VEL
LIN {X 0,Y 474.572,Z 246.866,A -85,B 0,C 180,E1 -7440.879,E2 -7440.879} C_VEL
LIN {X 0,Y 474.608,Z 246.869,A -85,B 0,C 180,E1 -7443.626,E2 -7443.626} C_VEL
LIN {X 0,Y 474.591,Z 246.863,A -85,B 0,C 180,E1 -7446.633,E2 -7446.633} C_VEL
LIN {X 0,Y 474.612,Z 246.864,A -85,B 0,C 180,E1 -7449.183,E2 -7449.183} C_VEL
LIN {X 0,Y 474.602,Z 246.867,A -85,B 0,C 180,E1 -7451.644,E2 -7451.644} C_VEL
LIN {X 0,Y 473.944,Z 246.949,A -85,B 0,C 180,E1 -7452.353,E2 -7452.353} C_VEL
LIN {X 0,Y 471.099,Z 247.308,A -85,B 0,C 180,E1 -7453.505,E2 -7453.505} C_VEL
LIN {X 0,Y 468.683,Z 247.609,A -85,B 0,C 180,E1 -7454.433,E2 -7454.433} C_VEL
LIN {X 0,Y 467.639,Z 247.737,A -85,B 0,C 180,E1 -7455.151,E2 -7455.151} C_VEL
LIN {X 0,Y 467.551,Z 247.746,A -85,B 0,C 180,E1 -7455.394,E2 -7455.394} C_VEL
LIN {X 0,Y 467.631,Z 247.734,A -85,B 0,C 180,E1 -7457.854,E2 -7457.854} C_VEL
LIN {X 0,Y 467.631,Z 247.738,A -85,B 0,C 180,E1 -7461.357,E2 -7461.357} C_VEL
LIN {X 0,Y 467.696,Z 247.726,A -85,B 0,C 180,E1 -7463.962,E2 -7463.962} C_VEL
LIN {X 0,Y 467.8,Z 247.716,A -85,B 0,C 180,E1 -7467.417,E2 -7467.417} C_VEL
LIN {X 0,Y 467.812,Z 247.712,A -85,B 0,C 180,E1 -7470,E2 -7470} C_VEL
LIN {X 0,Y 467.8,Z 247.716,A -85,B 0,C 180,E1 -7472.583,E2 -7472.583} C_VEL
LIN {X 0,Y 467.696,Z 247.726,A -85,B 0,C 180,E1 -7476.038,E2 -7476.038} C_VEL
LIN {X 0,Y 467.631,Z 247.738,A -85,B 0,C 180,E1 -7478.643,E2 -7478.643} C_VEL
LIN {X 0,Y 467.625,Z 247.736,A -85,B 0,C 180,E1 -7482.38,E2 -7482.38} C_VEL
LIN {X 0,Y 467.612,Z 247.737,A -85,B 0,C 180,E1 -7485.899,E2 -7485.899} C_VEL
LIN {X 0,Y 467.561,Z 247.739,A -85,B 0,C 180,E1 -7489.31,E2 -7489.31} C_VEL
LIN {X 0,Y 467.515,Z 247.748,A -85,B 0,C 180,E1 -7492.074,E2 -7492.074} C_VEL
LIN {X 0,Y 467.559,Z 247.741,A -85,B 0,C 180,E1 -7494.889,E2 -7494.889} C_VEL
LIN {X 0,Y 467.568,Z 247.74,A -85,B 0,C 180,E1 -7497.772,E2 -7497.772} C_VEL
LIN {X 0,Y 467.513,Z 247.745,A -85,B 0,C 180,E1 -7501.049,E2 -7501.049} C_VEL
LIN {X 0,Y 467.533,Z 247.749,A -85,B 0,C 180,E1 -7504.246,E2 -7504.246} C_VEL
LIN {X 0,Y 467.497,Z 247.747,A -85,B 0,C 180,E1 -7507.191,E2 -7507.191} C_VEL
LIN {X 0,Y 467.55,Z 247.745,A -85,B 0,C 180,E1 -7510.266,E2 -7510.266} C_VEL
LIN {X 0,Y 467.569,Z 247.739,A -85,B 0,C 180,E1 -7512.576,E2 -7512.576} C_VEL
LIN {X 0,Y 467.559,Z 247.742,A -85,B 0,C 180,E1 -7516.266,E2 -7516.266} C_VEL
LIN {X 0,Y 467.545,Z 247.741,A -85,B 0,C 180,E1 -7518.726,E2 -7518.726} C_VEL
LIN {X 0,Y 467.526,Z 247.748,A -85,B 0,C 180,E1 -7521.961,E2 -7521.961} C_VEL
LIN {X 0,Y 467.528,Z 247.746,A -85,B 0,C 180,E1 -7525.173,E2 -7525.173} C_VEL
LIN {X 0,Y 467.545,Z 247.742,A -85,B 0,C 180,E1 -7528.265,E2 -7528.265} C_VEL
LIN {X 0,Y 467.542,Z 247.747,A -85,B 0,C 180,E1 -7531.256,E2 -7531.256} C_VEL
LIN {X 0,Y 467.569,Z 247.738,A -85,B 0,C 180,E1 -7534.165,E2 -7534.165} C_VEL
LIN {X 0,Y 467.547,Z 247.745,A -85,B 0,C 180,E1 -7537.001,E2 -7537.001} C_VEL
LIN {X 0,Y 467.595,Z 247.737,A -85,B 0,C 180,E1 -7539.783,E2 -7539.783} C_VEL
LIN {X 0,Y 467.573,Z 247.738,A -85,B 0,C 180,E1 -7542.512,E2 -7542.512} C_VEL
LIN {X 0,Y 467.583,Z 247.744,A -85,B 0,C 180,E1 -7545.202,E2 -7545.202} C_VEL
LIN {X 0,Y 467.636,Z 247.73,A -85,B 0,C 180,E1 -7547.86,E2 -7547.86} C_VEL
LIN {X 0,Y 467.651,Z 247.731,A -85,B 0,C 180,E1 -7551.362,E2 -7551.362} C_VEL
LIN {X 0,Y 467.709,Z 247.721,A -85,B 0,C 180,E1 -7553.968,E2 -7553.968} C_VEL
LIN {X 0,Y 467.842,Z 247.705,A -85,B 0,C 180,E1 -7557.422,E2 -7557.422} C_VEL
LIN {X 0,Y 467.866,Z 247.701,A -85,B 0,C 180,E1 -7560.005,E2 -7560.005} C_VEL
LIN {X 0,Y 467.811,Z 247.715,A -85,B 0,C 180,E1 -7562.588,E2 -7562.588} C_VEL
LIN {X 0,Y 467.716,Z 247.721,A -85,B 0,C 180,E1 -7566.042,E2 -7566.042} C_VEL
LIN {X 0,Y 467.655,Z 247.734,A -85,B 0,C 180,E1 -7568.648,E2 -7568.648} C_VEL
LIN {X 0,Y 467.652,Z 247.732,A -85,B 0,C 180,E1 -7572.15,E2 -7572.15} C_VEL
LIN {X 0,Y 467.637,Z 247.73,A -85,B 0,C 180,E1 -7575.699,E2 -7575.699} C_VEL
LIN {X 0,Y 467.621,Z 247.732,A -85,B 0,C 180,E1 -7579.312,E2 -7579.312} C_VEL
LIN {X 0,Y 467.535,Z 247.748,A -85,B 0,C 180,E1 -7582.078,E2 -7582.078} C_VEL
LIN {X 0,Y 467.571,Z 247.738,A -85,B 0,C 180,E1 -7584.893,E2 -7584.893} C_VEL
LIN {X 0,Y 467.565,Z 247.743,A -85,B 0,C 180,E1 -7587.776,E2 -7587.776} C_VEL
LIN {X 0,Y 467.57,Z 247.738,A -85,B 0,C 180,E1 -7591.048,E2 -7591.048} C_VEL
LIN {X 0,Y 467.582,Z 247.743,A -85,B 0,C 180,E1 -7594.243,E2 -7594.243} C_VEL
LIN {X 0,Y 467.547,Z 247.745,A -85,B 0,C 180,E1 -7597.188,E2 -7597.188} C_VEL
LIN {X 0,Y 467.566,Z 247.746,A -85,B 0,C 180,E1 -7600.269,E2 -7600.269} C_VEL
LIN {X 0,Y 467.572,Z 247.745,A -85,B 0,C 180,E1 -7601.407,E2 -7601.407} C_VEL
LIN {X 0,Y 467.841,Z 249.946,A -85,B 0,C 180,E1 -7603.715,E2 -7603.715} C_VEL
LIN {X 0,Y 468.281,Z 253.051,A -85,B 0,C 180,E1 -7606.342,E2 -7606.342} C_VEL
LIN {X 0,Y 468.363,Z 256.065,A -85,B 0,C 180,E1 -7608.683,E2 -7608.683} C_VEL
LIN {X 0,Y 468.149,Z 260.69,A -85,B 0,C 180,E1 -7612.012,E2 -7612.012} C_VEL
LIN {X 0,Y 467.938,Z 265.451,A -85,B 0,C 180,E1 -7615.2,E2 -7615.2} C_VEL
LIN {X 0,Y 467.688,Z 270.285,A -85,B 0,C 180,E1 -7618.269,E2 -7618.269} C_VEL
LIN {X 0,Y 467.393,Z 275.23,A -85,B 0,C 180,E1 -7621.239,E2 -7621.239} C_VEL
LIN {X 0,Y 467.183,Z 280.894,A -85,B 0,C 180,E1 -7624.506,E2 -7624.506} C_VEL
LIN {X 0,Y 467.042,Z 285.312,A -85,B 0,C 180,E1 -7626.969,E2 -7626.969} C_VEL
LIN {X 0,Y 466.913,Z 290.451,A -85,B 0,C 180,E1 -7629.746,E2 -7629.746} C_VEL
LIN {X 0,Y 466.798,Z 295.625,A -85,B 0,C 180,E1 -7632.476,E2 -7632.476} C_VEL
LIN {X 0,Y 466.734,Z 299.787,A -85,B 0,C 180,E1 -7634.624,E2 -7634.624} C_VEL
LIN {X 0,Y 468.695,Z 311.253,A -85,B 0,C 180,E1 -7635.002,E2 -7635.002} C_VEL
LIN {X 0,Y 469.957,Z 320.181,A -85,B 0,C 180,E1 -7635.383,E2 -7635.383} C_VEL
LIN {X 0,Y 469.656,Z 329.258,A -85,B 0,C 180,E1 -7635.816,E2 -7635.816} C_VEL
LIN {X 0,Y 469.213,Z 338.391,A -85,B 0,C 180,E1 -7636.355,E2 -7636.355} C_VEL
LIN {X 0,Y 468.774,Z 347.389,A -85,B 0,C 180,E1 -7637.004,E2 -7637.004} C_VEL
LIN {X 0,Y 468.461,Z 355.486,A -85,B 0,C 180,E1 -7637.705,E2 -7637.705} C_VEL
LIN {X 0,Y 468.137,Z 363.519,A -85,B 0,C 180,E1 -7638.527,E2 -7638.527} C_VEL
LIN {X 0,Y 467.746,Z 370.739,A -85,B 0,C 180,E1 -7639.394,E2 -7639.394} C_VEL
LIN {X 0,Y 467.475,Z 376.942,A -85,B 0,C 180,E1 -7640.263,E2 -7640.263} C_VEL
LIN {X 0,Y 467.163,Z 383.479,A -85,B 0,C 180,E1 -7641.348,E2 -7641.348} C_VEL
LIN {X 0,Y 466.993,Z 387.98,A -85,B 0,C 180,E1 -7642.216,E2 -7642.216} C_VEL
LIN {X 0,Y 466.805,Z 393.628,A -85,B 0,C 180,E1 -7643.561,E2 -7643.561} C_VEL
LIN {X 0,Y 466.742,Z 397.793,A -85,B 0,C 180,E1 -7644.817,E2 -7644.817} C_VEL
LIN {X 0,Y 466.652,Z 400.156,A -85,B 0,C 180,E1 -7645.682,E2 -7645.682} C_VEL
LIN {X 0,Y 466.665,Z 401.953,A -85,B 0,C 180,E1 -7646.546,E2 -7646.546} C_VEL
LIN {X 0,Y 466.611,Z 404.393,A -85,B 0,C 180,E1 -7648.274,E2 -7648.274} C_VEL
LIN {X 0,Y 466.593,Z 404.98,A -85,B 0,C 180,E1 -7649.137,E2 -7649.137} C_VEL
LIN {X 0,Y 466.593,Z 404.98,A -85,B 0,C 180,E1 -7650.863,E2 -7650.863} C_VEL
LIN {X 0,Y 466.611,Z 404.393,A -85,B 0,C 180,E1 -7651.726,E2 -7651.726} C_VEL
LIN {X 0,Y 466.665,Z 401.953,A -85,B 0,C 180,E1 -7653.454,E2 -7653.454} C_VEL
LIN {X 0,Y 466.696,Z 399.008,A -85,B 0,C 180,E1 -7654.751,E2 -7654.751} C_VEL
LIN {X 0,Y 466.756,Z 395.022,A -85,B 0,C 180,E1 -7656.05,E2 -7656.05} C_VEL
LIN {X 0,Y 466.944,Z 389.896,A -85,B 0,C 180,E1 -7657.35,E2 -7657.35} C_VEL
LIN {X 0,Y 467.118,Z 384.634,A -85,B 0,C 180,E1 -7658.435,E2 -7658.435} C_VEL
LIN {X 0,Y 467.389,Z 378.318,A -85,B 0,C 180,E1 -7659.52,E2 -7659.52} C_VEL
LIN {X 0,Y 467.632,Z 372.365,A -85,B 0,C 180,E1 -7660.39,E2 -7660.39} C_VEL
LIN {X 0,Y 468.016,Z 365.438,A -85,B 0,C 180,E1 -7661.257,E2 -7661.257} C_VEL
LIN {X 0,Y 468.427,Z 357.257,A -85,B 0,C 180,E1 -7662.125,E2 -7662.125} C_VEL
LIN {X 0,Y 468.681,Z 349.796,A -85,B 0,C 180,E1 -7662.802,E2 -7662.802} C_VEL
LIN {X 0,Y 469.171,Z 340.024,A -85,B 0,C 180,E1 -7663.536,E2 -7663.536} C_VEL
LIN {X 0,Y 469.543,Z 330.263,A -85,B 0,C 180,E1 -7664.132,E2 -7664.132} C_VEL
LIN {X 0,Y 469.934,Z 321.47,A -85,B 0,C 180,E1 -7664.562,E2 -7664.562} C_VEL
LIN {X 0,Y 468.674,Z 311.252,A -85,B 0,C 180,E1 -7664.999,E2 -7664.999} C_VEL
LIN {X 0,Y 466.881,Z 301.135,A -85,B 0,C 180,E1 -7665.339,E2 -7665.339} C_VEL
LIN {X 0,Y 466.709,Z 299.743,A -85,B 0,C 180,E1 -7665.398,E2 -7665.398} C_VEL
LIN {X 0,Y 466.838,Z 293.786,A -85,B 0,C 180,E1 -7668.475,E2 -7668.475} C_VEL
LIN {X 0,Y 466.944,Z 288.72,A -85,B 0,C 180,E1 -7671.175,E2 -7671.175} C_VEL
LIN {X 0,Y 467.058,Z 283.611,A -85,B 0,C 180,E1 -7673.971,E2 -7673.971} C_VEL
LIN {X 0,Y 467.231,Z 278.554,A -85,B 0,C 180,E1 -7676.823,E2 -7676.823} C_VEL
LIN {X 0,Y 467.471,Z 273.565,A -85,B 0,C 180,E1 -7679.743,E2 -7679.743} C_VEL
LIN {X 0,Y 467.788,Z 268.656,A -85,B 0,C 180,E1 -7682.741,E2 -7682.741} C_VEL
LIN {X 0,Y 468.019,Z 263.835,A -85,B 0,C 180,E1 -7685.847,E2 -7685.847} C_VEL
LIN {X 0,Y 468.237,Z 259.125,A -85,B 0,C 180,E1 -7689.078,E2 -7689.078} C_VEL
LIN {X 0,Y 468.385,Z 255.943,A -85,B 0,C 180,E1 -7691.385,E2 -7691.385} C_VEL
LIN {X 0,Y 468.273,Z 252.724,A -85,B 0,C 180,E1 -7693.909,E2 -7693.909} C_VEL
LIN {X 0,Y 467.665,Z 248.654,A -85,B 0,C 180,E1 -7697.445,E2 -7697.445} C_VEL
LIN {X 0,Y 467.573,Z 247.744,A -85,B 0,C 180,E1 -7698.722,E2 -7698.722} C_VEL
LIN {X 0,Y 467.566,Z 247.745,A -85,B 0,C 180,E1 -7701.952,E2 -7701.952} C_VEL
LIN {X 0,Y 467.561,Z 247.743,A -85,B 0,C 180,E1 -7705.163,E2 -7705.163} C_VEL
LIN {X 0,Y 467.586,Z 247.741,A -85,B 0,C 180,E1 -7708.256,E2 -7708.256} C_VEL
LIN {X 0,Y 467.55,Z 247.741,A -85,B 0,C 180,E1 -7711.245,E2 -7711.245} C_VEL
LIN {X 0,Y 467.594,Z 247.737,A -85,B 0,C 180,E1 -7714.394,E2 -7714.394} C_VEL
LIN {X 0,Y 467.577,Z 247.737,A -85,B 0,C 180,E1 -7716.992,E2 -7716.992} C_VEL
LIN {X 0,Y 467.622,Z 247.739,A -85,B 0,C 180,E1 -7719.773,E2 -7719.773} C_VEL
LIN {X 0,Y 467.593,Z 247.735,A -85,B 0,C 180,E1 -7722.502,E2 -7722.502} C_VEL
LIN {X 0,Y 467.602,Z 247.737,A -85,B 0,C 180,E1 -7725.192,E2 -7725.192} C_VEL
LIN {X 0,Y 467.652,Z 247.732,A -85,B 0,C 180,E1 -7727.85,E2 -7727.85} C_VEL
LIN {X 0,Y 467.655,Z 247.734,A -85,B 0,C 180,E1 -7731.352,E2 -7731.352} C_VEL
LIN {X 0,Y 467.716,Z 247.721,A -85,B 0,C 180,E1 -7733.958,E2 -7733.958} C_VEL
LIN {X 0,Y 467.811,Z 247.715,A -85,B 0,C 180,E1 -7737.412,E2 -7737.412} C_VEL
LIN {X 0,Y 467.866,Z 247.701,A -85,B 0,C 180,E1 -7739.995,E2 -7739.995} C_VEL
LIN {X 0,Y 467.842,Z 247.705,A -85,B 0,C 180,E1 -7742.578,E2 -7742.578} C_VEL
LIN {X 0,Y 467.709,Z 247.721,A -85,B 0,C 180,E1 -7746.032,E2 -7746.032} C_VEL
LIN {X 0,Y 467.651,Z 247.731,A -85,B 0,C 180,E1 -7748.638,E2 -7748.638} C_VEL
LIN {X 0,Y 467.636,Z 247.73,A -85,B 0,C 180,E1 -7752.14,E2 -7752.14} C_VEL
LIN {X 0,Y 467.615,Z 247.732,A -85,B 0,C 180,E1 -7755.69,E2 -7755.69} C_VEL
LIN {X 0,Y 467.595,Z 247.736,A -85,B 0,C 180,E1 -7759.302,E2 -7759.302} C_VEL
LIN {X 0,Y 467.505,Z 247.747,A -85,B 0,C 180,E1 -7762.068,E2 -7762.068} C_VEL
LIN {X 0,Y 467.563,Z 247.743,A -85,B 0,C 180,E1 -7764.882,E2 -7764.882} C_VEL
LIN {X 0,Y 467.586,Z 247.736,A -85,B 0,C 180,E1 -7767.764,E2 -7767.764} C_VEL
LIN {X 0,Y 467.531,Z 247.744,A -85,B 0,C 180,E1 -7771.039,E2 -7771.039} C_VEL
LIN {X 0,Y 467.551,Z 247.746,A -85,B 0,C 180,E1 -7774.237,E2 -7774.237} C_VEL
LIN {X 0,Y 467.508,Z 247.746,A -85,B 0,C 180,E1 -7777.182,E2 -7777.182} C_VEL
LIN {X 0,Y 467.551,Z 247.748,A -85,B 0,C 180,E1 -7780.258,E2 -7780.258} C_VEL
LIN {X 0,Y 467.573,Z 247.741,A -85,B 0,C 180,E1 -7782.567,E2 -7782.567} C_VEL
LIN {X 0,Y 467.535,Z 247.742,A -85,B 0,C 180,E1 -7785.05,E2 -7785.05} C_VEL
LIN {X 0,Y 467.574,Z 247.739,A -85,B 0,C 180,E1 -7787.44,E2 -7787.44} C_VEL
LIN {X 0,Y 467.573,Z 247.738,A -85,B 0,C 180,E1 -7790.855,E2 -7790.855} C_VEL
LIN {X 0,Y 467.507,Z 247.749,A -85,B 0,C 180,E1 -7794.257,E2 -7794.257} C_VEL
LIN {X 0,Y 467.524,Z 247.746,A -85,B 0,C 180,E1 -7797.317,E2 -7797.317} C_VEL
LIN {X 0,Y 467.518,Z 247.744,A -85,B 0,C 180,E1 -7800.662,E2 -7800.662} C_VEL
LIN {X 0,Y 467.568,Z 247.741,A -85,B 0,C 180,E1 -7803.197,E2 -7803.197} C_VEL
LIN {X 0,Y 467.531,Z 247.745,A -85,B 0,C 180,E1 -7806.055,E2 -7806.055} C_VEL
LIN {X 0,Y 467.577,Z 247.738,A -85,B 0,C 180,E1 -7808.855,E2 -7808.855} C_VEL
LIN {X 0,Y 467.574,Z 247.744,A -85,B 0,C 180,E1 -7811.635,E2 -7811.635} C_VEL
LIN {X 0,Y 467.603,Z 247.737,A -85,B 0,C 180,E1 -7814.304,E2 -7814.304} C_VEL
LIN {X 0,Y 467.551,Z 247.746,A -85,B 0,C 180,E1 -7815.394,E2 -7815.394} C_VEL
LIN {X 0,Y 466.88,Z 247.828,A -85,B 0,C 180,E1 -7816.113,E2 -7816.113} C_VEL
LIN {X 0,Y 464.041,Z 248.186,A -85,B 0,C 180,E1 -7817.282,E2 -7817.282} C_VEL
LIN {X 0,Y 461.644,Z 248.48,A -85,B 0,C 180,E1 -7818.225,E2 -7818.225} C_VEL
LIN {X 0,Y 460.614,Z 248.611,A -85,B 0,C 180,E1 -7818.953,E2 -7818.953} C_VEL
LIN {X 0,Y 460.529,Z 248.619,A -85,B 0,C 180,E1 -7819.199,E2 -7819.199} C_VEL
LIN {X 0,Y 460.663,Z 248.603,A -85,B 0,C 180,E1 -7822.528,E2 -7822.528} C_VEL
LIN {X 0,Y 460.643,Z 248.606,A -85,B 0,C 180,E1 -7824.748,E2 -7824.748} C_VEL
LIN {X 0,Y 460.766,Z 248.592,A -85,B 0,C 180,E1 -7827.377,E2 -7827.377} C_VEL
LIN {X 0,Y 460.784,Z 248.588,A -85,B 0,C 180,E1 -7830,E2 -7830} C_VEL
LIN {X 0,Y 460.766,Z 248.592,A -85,B 0,C 180,E1 -7832.623,E2 -7832.623} C_VEL
LIN {X 0,Y 460.661,Z 248.603,A -85,B 0,C 180,E1 -7836.13,E2 -7836.13} C_VEL
LIN {X 0,Y 460.598,Z 248.614,A -85,B 0,C 180,E1 -7838.776,E2 -7838.776} C_VEL
LIN {X 0,Y 460.568,Z 248.616,A -85,B 0,C 180,E1 -7842.458,E2 -7842.458} C_VEL
LIN {X 0,Y 460.557,Z 248.616,A -85,B 0,C 180,E1 -7846.009,E2 -7846.009} C_VEL
LIN {X 0,Y 460.511,Z 248.62,A -85,B 0,C 180,E1 -7848.906,E2 -7848.906} C_VEL
LIN {X 0,Y 460.501,Z 248.618,A -85,B 0,C 180,E1 -7851.486,E2 -7851.486} C_VEL
LIN {X 0,Y 460.497,Z 248.626,A -85,B 0,C 180,E1 -7854.334,E2 -7854.334} C_VEL
LIN {X 0,Y 460.524,Z 248.616,A -85,B 0,C 180,E1 -7857.246,E2 -7857.246} C_VEL
LIN {X 0,Y 460.468,Z 248.631,A -85,B 0,C 180,E1 -7860.242,E2 -7860.242} C_VEL
LIN {X 0,Y 460.472,Z 248.622,A -85,B 0,C 180,E1 -7863.329,E2 -7863.329} C_VEL
LIN {X 0,Y 460.424,Z 248.631,A -85,B 0,C 180,E1 -7866.533,E2 -7866.533} C_VEL
LIN {X 0,Y 460.534,Z 248.62,A -85,B 0,C 180,E1 -7869.861,E2 -7869.861} C_VEL
LIN {X 0,Y 460.492,Z 248.62,A -85,B 0,C 180,E1 -7872.909,E2 -7872.909} C_VEL
LIN {X 0,Y 460.5,Z 248.626,A -85,B 0,C 180,E1 -7875.83,E2 -7875.83} C_VEL
LIN {X 0,Y 460.498,Z 248.619,A -85,B 0,C 180,E1 -7878.995,E2 -7878.995} C_VEL
LIN {X 0,Y 460.495,Z 248.622,A -85,B 0,C 180,E1 -7881.273,E2 -7881.273} C_VEL
LIN {X 0,Y 460.473,Z 248.622,A -85,B 0,C 180,E1 -7884.56,E2 -7884.56} C_VEL
LIN {X 0,Y 460.493,Z 248.625,A -85,B 0,C 180,E1 -7887.721,E2 -7887.721} C_VEL
LIN {X 0,Y 460.504,Z 248.619,A -85,B 0,C 180,E1 -7890.774,E2 -7890.774} C_VEL
LIN {X 0,Y 460.526,Z 248.619,A -85,B 0,C 180,E1 -7893.74,E2 -7893.74} C_VEL
LIN {X 0,Y 460.516,Z 248.617,A -85,B 0,C 180,E1 -7896.629,E2 -7896.629} C_VEL
LIN {X 0,Y 460.524,Z 248.621,A -85,B 0,C 180,E1 -7899.458,E2 -7899.458} C_VEL
LIN {X 0,Y 460.524,Z 248.616,A -85,B 0,C 180,E1 -7902.235,E2 -7902.235} C_VEL
LIN {X 0,Y 460.542,Z 248.619,A -85,B 0,C 180,E1 -7904.97,E2 -7904.97} C_VEL
LIN {X 0,Y 460.591,Z 248.61,A -85,B 0,C 180,E1 -7908.565,E2 -7908.565} C_VEL
LIN {X 0,Y 460.601,Z 248.611,A -85,B 0,C 180,E1 -7911.229,E2 -7911.229} C_VEL
LIN {X 0,Y 460.675,Z 248.597,A -85,B 0,C 180,E1 -7913.875,E2 -7913.875} C_VEL
LIN {X 0,Y 460.784,Z 248.585,A -85,B 0,C 180,E1 -7917.383,E2 -7917.383} C_VEL
LIN {X 0,Y 460.837,Z 248.577,A -85,B 0,C 180,E1 -7920.005,E2 -7920.005} C_VEL
LIN {X 0,Y 460.755,Z 248.594,A -85,B 0,C 180,E1 -7922.628,E2 -7922.628} C_VEL
LIN {X 0,Y 460.682,Z 248.598,A -85,B 0,C 180,E1 -7926.135,E2 -7926.135} C_VEL
LIN {X 0,Y 460.606,Z 248.61,A -85,B 0,C 180,E1 -7928.781,E2 -7928.781} C_VEL
LIN {X 0,Y 460.606,Z 248.612,A -85,B 0,C 180,E1 -7932.339,E2 -7932.339} C_VEL
LIN {X 0,Y 460.6,Z 248.61,A -85,B 0,C 180,E1 -7936.002,E2 -7936.002} C_VEL
LIN {X 0,Y 460.567,Z 248.611,A -85,B 0,C 180,E1 -7939.62,E2 -7939.62} C_VEL
LIN {X 0,Y 460.512,Z 248.622,A -85,B 0,C 180,E1 -7942.433,E2 -7942.433} C_VEL
LIN {X 0,Y 460.547,Z 248.617,A -85,B 0,C 180,E1 -7945.799,E2 -7945.799} C_VEL
LIN {X 0,Y 460.519,Z 248.622,A -85,B 0,C 180,E1 -7948.239,E2 -7948.239} C_VEL
LIN {X 0,Y 460.525,Z 248.616,A -85,B 0,C 180,E1 -7951.286,E2 -7951.286} C_VEL
LIN {X 0,Y 460.527,Z 248.618,A -85,B 0,C 180,E1 -7954.507,E2 -7954.507} C_VEL
LIN {X 0,Y 460.504,Z 248.626,A -85,B 0,C 180,E1 -7957.627,E2 -7957.627} C_VEL
LIN {X 0,Y 460.526,Z 248.623,A -85,B 0,C 180,E1 -7961.015,E2 -7961.015} C_VEL
LIN {X 0,Y 460.539,Z 248.805,A -85,B 0,C 180,E1 -7961.605,E2 -7961.605} C_VEL
LIN {X 0,Y 461.003,Z 252.038,A -85,B 0,C 180,E1 -7964.533,E2 -7964.533} C_VEL
LIN {X 0,Y 461.31,Z 254.977,A -85,B 0,C 180,E1 -7966.997,E2 -7966.997} C_VEL
LIN {X 0,Y 461.271,Z 258.398,A -85,B 0,C 180,E1 -7969.628,E2 -7969.628} C_VEL
LIN {X 0,Y 461.113,Z 262.288,A -85,B 0,C 180,E1 -7972.437,E2 -7972.437} C_VEL
LIN {X 0,Y 460.872,Z 267.06,A -85,B 0,C 180,E1 -7975.652,E2 -7975.652} C_VEL
LIN {X 0,Y 460.573,Z 271.911,A -85,B 0,C 180,E1 -7978.748,E2 -7978.748} C_VEL
LIN {X 0,Y 460.285,Z 276.845,A -85,B 0,C 180,E1 -7981.75,E2 -7981.75} C_VEL
LIN {X 0,Y 460.113,Z 281.854,A -85,B 0,C 180,E1 -7984.68,E2 -7984.68} C_VEL
LIN {X 0,Y 459.902,Z 286.915,A -85,B 0,C 180,E1 -7987.541,E2 -7987.541} C_VEL
LIN {X 0,Y 459.796,Z 292.028,A -85,B 0,C 180,E1 -7990.351,E2 -7990.351} C_VEL
LIN {X 0,Y 459.691,Z 297.186,A -85,B 0,C 180,E1 -7993.114,E2 -7993.114} C_VEL
LIN {X 0,Y 459.649,Z 299.614,A -85,B 0,C 180,E1 -7994.374,E2 -7994.374} C_VEL
LIN {X 0,Y 462.031,Z 313.691,A -85,B 0,C 180,E1 -7994.865,E2 -7994.865} C_VEL
LIN {X 0,Y 462.994,Z 322.562,A -85,B 0,C 180,E1 -7995.271,E2 -7995.271} C_VEL
LIN {X 0,Y 462.469,Z 334.93,A -85,B 0,C 180,E1 -7995.928,E2 -7995.928} C_VEL
LIN {X 0,Y 461.927,Z 345.842,A -85,B 0,C 180,E1 -7996.696,E2 -7996.696} C_VEL
LIN {X 0,Y 461.486,Z 355.471,A -85,B 0,C 180,E1 -7997.534,E2 -7997.534} C_VEL
LIN {X 0,Y 461.142,Z 363.324,A -85,B 0,C 180,E1 -7998.35,E2 -7998.35} C_VEL
LIN {X 0,Y 460.737,Z 370.543,A -85,B 0,C 180,E1 -7999.231,E2 -7999.231} C_VEL
LIN {X 0,Y 460.462,Z 376.747,A -85,B 0,C 180,E1 -8000.113,E2 -8000.113} C_VEL
LIN {X 0,Y 460.124,Z 383.283,A -85,B 0,C 180,E1 -8001.214,E2 -8001.214} C_VEL
LIN {X 0,Y 459.913,Z 387.784,A -85,B 0,C 180,E1 -8002.095,E2 -8002.095} C_VEL
LIN {X 0,Y 459.752,Z 392.768,A -85,B 0,C 180,E1 -8003.273,E2 -8003.273} C_VEL
LIN {X 0,Y 459.656,Z 397.598,A -85,B 0,C 180,E1 -8004.737,E2 -8004.737} C_VEL
LIN {X 0,Y 459.57,Z 399.961,A -85,B 0,C 180,E1 -8005.615,E2 -8005.615} C_VEL
LIN {X 0,Y 459.562,Z 401.758,A -85,B 0,C 180,E1 -8006.493,E2 -8006.493} C_VEL
LIN {X 0,Y 459.524,Z 404.198,A -85,B 0,C 180,E1 -8008.247,E2 -8008.247} C_VEL
LIN {X 0,Y 459.499,Z 404.785,A -85,B 0,C 180,E1 -8009.124,E2 -8009.124} C_VEL
LIN {X 0,Y 459.499,Z 404.785,A -85,B 0,C 180,E1 -8010.876,E2 -8010.876} C_VEL
LIN {X 0,Y 459.524,Z 404.198,A -85,B 0,C 180,E1 -8011.753,E2 -8011.753} C_VEL
LIN {X 0,Y 459.562,Z 401.758,A -85,B 0,C 180,E1 -8013.507,E2 -8013.507} C_VEL
LIN {X 0,Y 459.623,Z 398.813,A -85,B 0,C 180,E1 -8014.824,E2 -8014.824} C_VEL
LIN {X 0,Y 459.667,Z 394.827,A -85,B 0,C 180,E1 -8016.144,E2 -8016.144} C_VEL
LIN {X 0,Y 459.864,Z 389.7,A -85,B 0,C 180,E1 -8017.464,E2 -8017.464} C_VEL
LIN {X 0,Y 460.053,Z 384.439,A -85,B 0,C 180,E1 -8018.566,E2 -8018.566} C_VEL
LIN {X 0,Y 460.373,Z 378.122,A -85,B 0,C 180,E1 -8019.667,E2 -8019.667} C_VEL
LIN {X 0,Y 460.616,Z 372.169,A -85,B 0,C 180,E1 -8020.55,E2 -8020.55} C_VEL
LIN {X 0,Y 461.029,Z 365.243,A -85,B 0,C 180,E1 -8021.43,E2 -8021.43} C_VEL
LIN {X 0,Y 461.458,Z 357.062,A -85,B 0,C 180,E1 -8022.311,E2 -8022.311} C_VEL
LIN {X 0,Y 461.748,Z 348.855,A -85,B 0,C 180,E1 -8023.059,E2 -8023.059} C_VEL
LIN {X 0,Y 462.249,Z 339.829,A -85,B 0,C 180,E1 -8023.742,E2 -8023.742} C_VEL
LIN {X 0,Y 462.609,Z 331.075,A -85,B 0,C 180,E1 -8024.292,E2 -8024.292} C_VEL
LIN {X 0,Y 463.04,Z 321.274,A -85,B 0,C 180,E1 -8024.784,E2 -8024.784} C_VEL
LIN {X 0,Y 461.558,Z 310.598,A -85,B 0,C 180,E1 -8025.25,E2 -8025.25} C_VEL
LIN {X 0,Y 459.649,Z 299.614,A -85,B 0,C 180,E1 -8025.626,E2 -8025.626} C_VEL
LIN {X 0,Y 459.755,Z 293.74,A -85,B 0,C 180,E1 -8028.724,E2 -8028.724} C_VEL
LIN {X 0,Y 459.869,Z 288.612,A -85,B 0,C 180,E1 -8031.517,E2 -8031.517} C_VEL
LIN {X 0,Y 460.013,Z 283.527,A -85,B 0,C 180,E1 -8034.361,E2 -8034.361} C_VEL
LIN {X 0,Y 460.213,Z 278.497,A -85,B 0,C 180,E1 -8037.266,E2 -8037.266} C_VEL
LIN {X 0,Y 460.469,Z 273.536,A -85,B 0,C 180,E1 -8040.242,E2 -8040.242} C_VEL
LIN {X 0,Y 460.753,Z 268.651,A -85,B 0,C 180,E1 -8043.306,E2 -8043.306} C_VEL
LIN {X 0,Y 461.008,Z 263.861,A -85,B 0,C 180,E1 -8046.479,E2 -8046.479} C_VEL
LIN {X 0,Y 461.247,Z 259.179,A -85,B 0,C 180,E1 -8049.787,E2 -8049.787} C_VEL
LIN {X 0,Y 461.357,Z 256.118,A -85,B 0,C 180,E1 -8052.086,E2 -8052.086} C_VEL
LIN {X 0,Y 461.166,Z 253.138,A -85,B 0,C 180,E1 -8054.508,E2 -8054.508} C_VEL
LIN {X 0,Y 460.609,Z 249.415,A -85,B 0,C 180,E1 -8057.825,E2 -8057.825} C_VEL
LIN {X 0,Y 460.539,Z 248.804,A -85,B 0,C 180,E1 -8058.395,E2 -8058.395} C_VEL
LIN {X 0,Y 460.52,Z 248.621,A -85,B 0,C 180,E1 -8061.263,E2 -8061.263} C_VEL
LIN {X 0,Y 460.511,Z 248.624,A -85,B 0,C 180,E1 -8064.551,E2 -8064.551} C_VEL
LIN {X 0,Y 460.535,Z 248.618,A -85,B 0,C 180,E1 -8067.712,E2 -8067.712} C_VEL
LIN {X 0,Y 460.526,Z 248.616,A -85,B 0,C 180,E1 -8070.764,E2 -8070.764} C_VEL
LIN {X 0,Y 460.527,Z 248.621,A -85,B 0,C 180,E1 -8073.729,E2 -8073.729} C_VEL
LIN {X 0,Y 460.546,Z 248.613,A -85,B 0,C 180,E1 -8076.62,E2 -8076.62} C_VEL
LIN {X 0,Y 460.551,Z 248.616,A -85,B 0,C 180,E1 -8079.449,E2 -8079.449} C_VEL
LIN {X 0,Y 460.545,Z 248.615,A -85,B 0,C 180,E1 -8082.225,E2 -8082.225} C_VEL
LIN {X 0,Y 460.562,Z 248.612,A -85,B 0,C 180,E1 -8084.96,E2 -8084.96} C_VEL
LIN {X 0,Y 460.604,Z 248.606,A -85,B 0,C 180,E1 -8088.555,E2 -8088.555} C_VEL
LIN {X 0,Y 460.606,Z 248.61,A -85,B 0,C 180,E1 -8091.219,E2 -8091.219} C_VEL
LIN {X 0,Y 460.682,Z 248.598,A -85,B 0,C 180,E1 -8093.865,E2 -8093.865} C_VEL
LIN {X 0,Y 460.755,Z 248.594,A -85,B 0,C 180,E1 -8097.372,E2 -8097.372} C_VEL
LIN {X 0,Y 460.837,Z 248.577,A -85,B 0,C 180,E1 -8099.995,E2 -8099.995} C_VEL
LIN {X 0,Y 460.784,Z 248.585,A -85,B 0,C 180,E1 -8102.617,E2 -8102.617} C_VEL
LIN {X 0,Y 460.675,Z 248.597,A -85,B 0,C 180,E1 -8106.125,E2 -8106.125} C_VEL
LIN {X 0,Y 460.601,Z 248.611,A -85,B 0,C 180,E1 -8108.771,E2 -8108.771} C_VEL
LIN {X 0,Y 460.594,Z 248.609,A -85,B 0,C 180,E1 -8112.439,E2 -8112.439} C_VEL
LIN {X 0,Y 460.577,Z 248.609,A -85,B 0,C 180,E1 -8115.992,E2 -8115.992} C_VEL
LIN {X 0,Y 460.541,Z 248.614,A -85,B 0,C 180,E1 -8119.61,E2 -8119.61} C_VEL
LIN {X 0,Y 460.481,Z 248.626,A -85,B 0,C 180,E1 -8122.423,E2 -8122.423} C_VEL
LIN {X 0,Y 460.525,Z 248.616,A -85,B 0,C 180,E1 -8125.794,E2 -8125.794} C_VEL
LIN {X 0,Y 460.518,Z 248.62,A -85,B 0,C 180,E1 -8128.228,E2 -8128.228} C_VEL
LIN {X 0,Y 460.483,Z 248.621,A -85,B 0,C 180,E1 -8131.277,E2 -8131.277} C_VEL
LIN {X 0,Y 460.494,Z 248.626,A -85,B 0,C 180,E1 -8134.501,E2 -8134.501} C_VEL
LIN {X 0,Y 460.487,Z 248.621,A -85,B 0,C 180,E1 -8137.615,E2 -8137.615} C_VEL
LIN {X 0,Y 460.514,Z 248.625,A -85,B 0,C 180,E1 -8140.267,E2 -8140.267} C_VEL
LIN {X 0,Y 460.498,Z 248.619,A -85,B 0,C 180,E1 -8143.365,E2 -8143.365} C_VEL
LIN {X 0,Y 460.475,Z 248.624,A -85,B 0,C 180,E1 -8146.623,E2 -8146.623} C_VEL
LIN {X 0,Y 460.512,Z 248.621,A -85,B 0,C 180,E1 -8149.723,E2 -8149.723} C_VEL
LIN {X 0,Y 460.474,Z 248.623,A -85,B 0,C 180,E1 -8152.515,E2 -8152.515} C_VEL
LIN {X 0,Y 460.492,Z 248.625,A -85,B 0,C 180,E1 -8155.62,E2 -8155.62} C_VEL
LIN {X 0,Y 460.479,Z 248.621,A -85,B 0,C 180,E1 -8158.741,E2 -8158.741} C_VEL
LIN {X 0,Y 460.498,Z 248.626,A -85,B 0,C 180,E1 -8161.764,E2 -8161.764} C_VEL
LIN {X 0,Y 460.524,Z 248.616,A -85,B 0,C 180,E1 -8164.704,E2 -8164.704} C_VEL
LIN {X 0,Y 460.478,Z 248.629,A -85,B 0,C 180,E1 -8167.57,E2 -8167.57} C_VEL
LIN {X 0,Y 460.507,Z 248.618,A -85,B 0,C 180,E1 -8170.382,E2 -8170.382} C_VEL
LIN {X 0,Y 460.511,Z 248.624,A -85,B 0,C 180,E1 -8173.145,E2 -8173.145} C_VEL
LIN {X 0,Y 460.507,Z 248.623,A -85,B 0,C 180,E1 -8175.867,E2 -8175.867} C_VEL
LIN {X 0,Y 460.571,Z 248.613,A -85,B 0,C 180,E1 -8178.559,E2 -8178.559} C_VEL
LIN {X 0,Y 460.529,Z 248.619,A -85,B 0,C 180,E1 -8179.199,E2 -8179.199} C_VEL
LIN {X 0,Y 459.867,Z 248.706,A -85,B 0,C 180,E1 -8179.929,E2 -8179.929} C_VEL
LIN {X 0,Y 457.048,Z 249.061,A -85,B 0,C 180,E1 -8181.116,E2 -8181.116} C_VEL
LIN {X 0,Y 454.673,Z 249.355,A -85,B 0,C 180,E1 -8182.073,E2 -8182.073} C_VEL
LIN {X 0,Y 453.662,Z 249.478,A -85,B 0,C 180,E1 -8182.812,E2 -8182.812} C_VEL
LIN {X 0,Y 453.585,Z 249.485,A -85,B 0,C 180,E1 -8183.062,E2 -8183.062} C_VEL
LIN {X 0,Y 453.616,Z 249.481,A -85,B 0,C 180,E1 -8184.666,E2 -8184.666} C_VEL
LIN {X 0,Y 453.707,Z 249.472,A -85,B 0,C 180,E1 -8187.337,E2 -8187.337} C_VEL
LIN {X 0,Y 453.755,Z 249.463,A -85,B 0,C 180,E1 -8190,E2 -8190} C_VEL
LIN {X 0,Y 453.707,Z 249.472,A -85,B 0,C 180,E1 -8192.663,E2 -8192.663} C_VEL
LIN {X 0,Y 453.628,Z 249.479,A -85,B 0,C 180,E1 -8196.226,E2 -8196.226} C_VEL
LIN {X 0,Y 453.553,Z 249.491,A -85,B 0,C 180,E1 -8198.914,E2 -8198.914} C_VEL
LIN {X 0,Y 453.536,Z 249.493,A -85,B 0,C 180,E1 -8202.552,E2 -8202.552} C_VEL
LIN {X 0,Y 453.493,Z 249.497,A -85,B 0,C 180,E1 -8206.197,E2 -8206.197} C_VEL
LIN {X 0,Y 453.46,Z 249.498,A -85,B 0,C 180,E1 -8209.044,E2 -8209.044} C_VEL
LIN {X 0,Y 453.442,Z 249.499,A -85,B 0,C 180,E1 -8211.837,E2 -8211.837} C_VEL
LIN {X 0,Y 453.471,Z 249.498,A -85,B 0,C 180,E1 -8214.736,E2 -8214.736} C_VEL
LIN {X 0,Y 453.478,Z 249.497,A -85,B 0,C 180,E1 -8217.964,E2 -8217.964} C_VEL
LIN {X 0,Y 453.425,Z 249.502,A -85,B 0,C 180,E1 -8220.763,E2 -8220.763} C_VEL
LIN {X 0,Y 453.421,Z 249.505,A -85,B 0,C 180,E1 -8223.916,E2 -8223.916} C_VEL
LIN {X 0,Y 453.418,Z 249.501,A -85,B 0,C 180,E1 -8227.192,E2 -8227.192} C_VEL
LIN {X 0,Y 453.486,Z 249.494,A -85,B 0,C 180,E1 -8229.449,E2 -8229.449} C_VEL
LIN {X 0,Y 453.442,Z 249.498,A -85,B 0,C 180,E1 -8232.996,E2 -8232.996} C_VEL
LIN {X 0,Y 453.477,Z 249.501,A -85,B 0,C 180,E1 -8235.791,E2 -8235.791} C_VEL
LIN {X 0,Y 453.472,Z 249.497,A -85,B 0,C 180,E1 -8239.411,E2 -8239.411} C_VEL
LIN {X 0,Y 453.433,Z 249.501,A -85,B 0,C 180,E1 -8242.228,E2 -8242.228} C_VEL
LIN {X 0,Y 453.449,Z 249.5,A -85,B 0,C 180,E1 -8245.228,E2 -8245.228} C_VEL
LIN {X 0,Y 453.428,Z 249.5,A -85,B 0,C 180,E1 -8248.481,E2 -8248.481} C_VEL
LIN {X 0,Y 453.498,Z 249.492,A -85,B 0,C 180,E1 -8252.046,E2 -8252.046} C_VEL
LIN {X 0,Y 453.476,Z 249.5,A -85,B 0,C 180,E1 -8255.271,E2 -8255.271} C_VEL
LIN {X 0,Y 453.452,Z 249.497,A -85,B 0,C 180,E1 -8258.421,E2 -8258.421} C_VEL
LIN {X 0,Y 453.496,Z 249.496,A -85,B 0,C 180,E1 -8261.014,E2 -8261.014} C_VEL
LIN {X 0,Y 453.546,Z 249.486,A -85,B 0,C 180,E1 -8263.885,E2 -8263.885} C_VEL
LIN {X 0,Y 453.544,Z 249.488,A -85,B 0,C 180,E1 -8267.477,E2 -8267.477} C_VEL
LIN {X 0,Y 453.567,Z 249.489,A -85,B 0,C 180,E1 -8271.092,E2 -8271.092} C_VEL
LIN {X 0,Y 453.643,Z 249.473,A -85,B 0,C 180,E1 -8273.78,E2 -8273.78} C_VEL
LIN {X 0,Y 453.728,Z 249.464,A -85,B 0,C 180,E1 -8277.342,E2 -8277.342} C_VEL
LIN {X 0,Y 453.807,Z 249.453,A -85,B 0,C 180,E1 -8280.005,E2 -8280.005} C_VEL
LIN {X 0,Y 453.702,Z 249.473,A -85,B 0,C 180,E1 -8282.669,E2 -8282.669} C_VEL
LIN {X 0,Y 453.649,Z 249.475,A -85,B 0,C 180,E1 -8286.231,E2 -8286.231} C_VEL
LIN {X 0,Y 453.573,Z 249.485,A -85,B 0,C 180,E1 -8288.918,E2 -8288.918} C_VEL
LIN {X 0,Y 453.562,Z 249.49,A -85,B 0,C 180,E1 -8292.533,E2 -8292.533} C_VEL
LIN {X 0,Y 453.544,Z 249.491,A -85,B 0,C 180,E1 -8296.2,E2 -8296.2} C_VEL
LIN {X 0,Y 453.517,Z 249.489,A -85,B 0,C 180,E1 -8299.043,E2 -8299.043} C_VEL
LIN {X 0,Y 453.478,Z 249.497,A -85,B 0,C 180,E1 -8301.84,E2 -8301.84} C_VEL
LIN {X 0,Y 453.496,Z 249.493,A -85,B 0,C 180,E1 -8304.74,E2 -8304.74} C_VEL
LIN {X 0,Y 453.479,Z 249.5,A -85,B 0,C 180,E1 -8307.949,E2 -8307.949} C_VEL
LIN {X 0,Y 453.479,Z 249.494,A -85,B 0,C 180,E1 -8310.763,E2 -8310.763} C_VEL
LIN {X 0,Y 453.473,Z 249.502,A -85,B 0,C 180,E1 -8313.917,E2 -8313.917} C_VEL
LIN {X 0,Y 453.455,Z 249.501,A -85,B 0,C 180,E1 -8317.193,E2 -8317.193} C_VEL
LIN {X 0,Y 453.478,Z 249.5,A -85,B 0,C 180,E1 -8320.614,E2 -8320.614} C_VEL
LIN {X 0,Y 453.599,Z 250.357,A -85,B 0,C 180,E1 -8321.954,E2 -8321.954} C_VEL
LIN {X 0,Y 454.149,Z 254.155,A -85,B 0,C 180,E1 -8325.39,E2 -8325.39} C_VEL
LIN {X 0,Y 454.346,Z 257.715,A -85,B 0,C 180,E1 -8328.308,E2 -8328.308} C_VEL
LIN {X 0,Y 454.116,Z 262.341,A -85,B 0,C 180,E1 -8331.754,E2 -8331.754} C_VEL
LIN {X 0,Y 453.936,Z 265.464,A -85,B 0,C 180,E1 -8333.962,E2 -8333.962} C_VEL
LIN {X 0,Y 453.686,Z 270.279,A -85,B 0,C 180,E1 -8337.169,E2 -8337.169} C_VEL
LIN {X 0,Y 453.381,Z 275.147,A -85,B 0,C 180,E1 -8340.262,E2 -8340.262} C_VEL
LIN {X 0,Y 453.11,Z 280.104,A -85,B 0,C 180,E1 -8343.269,E2 -8343.269} C_VEL
LIN {X 0,Y 452.927,Z 285.26,A -85,B 0,C 180,E1 -8346.281,E2 -8346.281} C_VEL
LIN {X 0,Y 452.766,Z 290.209,A -85,B 0,C 180,E1 -8349.084,E2 -8349.084} C_VEL
LIN {X 0,Y 452.638,Z 295.314,A -85,B 0,C 180,E1 -8351.909,E2 -8351.909} C_VEL
LIN {X 0,Y 452.567,Z 299.484,A -85,B 0,C 180,E1 -8354.137,E2 -8354.137} C_VEL
LIN {X 0,Y 454.331,Z 309.217,A -85,B 0,C 180,E1 -8354.463,E2 -8354.463} C_VEL
LIN {X 0,Y 455.66,Z 318.486,A -85,B 0,C 180,E1 -8354.857,E2 -8354.857} C_VEL
LIN {X 0,Y 456.067,Z 323.653,A -85,B 0,C 180,E1 -8355.099,E2 -8355.099} C_VEL
LIN {X 0,Y 455.486,Z 336.369,A -85,B 0,C 180,E1 -8355.822,E2 -8355.822} C_VEL
LIN {X 0,Y 455.009,Z 345.647,A -85,B 0,C 180,E1 -8356.49,E2 -8356.49} C_VEL
LIN {X 0,Y 454.588,Z 354.104,A -85,B 0,C 180,E1 -8357.224,E2 -8357.224} C_VEL
LIN {X 0,Y 454.135,Z 363.127,A -85,B 0,C 180,E1 -8358.168,E2 -8358.168} C_VEL
LIN {X 0,Y 453.706,Z 370.347,A -85,B 0,C 180,E1 -8359.062,E2 -8359.062} C_VEL
LIN {X 0,Y 453.434,Z 376.551,A -85,B 0,C 180,E1 -8359.958,E2 -8359.958} C_VEL
LIN {X 0,Y 453.051,Z 383.087,A -85,B 0,C 180,E1 -8361.076,E2 -8361.076} C_VEL
LIN {X 0,Y 452.86,Z 387.589,A -85,B 0,C 180,E1 -8361.971,E2 -8361.971} C_VEL
LIN {X 0,Y 452.656,Z 393.235,A -85,B 0,C 180,E1 -8363.358,E2 -8363.358} C_VEL
LIN {X 0,Y 452.57,Z 397.402,A -85,B 0,C 180,E1 -8364.654,E2 -8364.654} C_VEL
LIN {X 0,Y 452.492,Z 399.766,A -85,B 0,C 180,E1 -8365.546,E2 -8365.546} C_VEL
LIN {X 0,Y 452.46,Z 401.563,A -85,B 0,C 180,E1 -8366.438,E2 -8366.438} C_VEL
LIN {X 0,Y 452.441,Z 404.004,A -85,B 0,C 180,E1 -8368.22,E2 -8368.22} C_VEL
LIN {X 0,Y 452.408,Z 404.591,A -85,B 0,C 180,E1 -8369.11,E2 -8369.11} C_VEL
LIN {X 0,Y 452.408,Z 404.591,A -85,B 0,C 180,E1 -8370.89,E2 -8370.89} C_VEL
LIN {X 0,Y 452.441,Z 404.004,A -85,B 0,C 180,E1 -8371.78,E2 -8371.78} C_VEL
LIN {X 0,Y 452.46,Z 401.563,A -85,B 0,C 180,E1 -8373.562,E2 -8373.562} C_VEL
LIN {X 0,Y 452.551,Z 398.619,A -85,B 0,C 180,E1 -8374.9,E2 -8374.9} C_VEL
LIN {X 0,Y 452.595,Z 394.632,A -85,B 0,C 180,E1 -8376.24,E2 -8376.24} C_VEL
LIN {X 0,Y 452.792,Z 389.505,A -85,B 0,C 180,E1 -8377.581,E2 -8377.581} C_VEL
LIN {X 0,Y 453.012,Z 384.243,A -85,B 0,C 180,E1 -8378.7,E2 -8378.7} C_VEL
LIN {X 0,Y 453.345,Z 377.927,A -85,B 0,C 180,E1 -8379.818,E2 -8379.818} C_VEL
LIN {X 0,Y 453.608,Z 371.974,A -85,B 0,C 180,E1 -8380.715,E2 -8380.715} C_VEL
LIN {X 0,Y 454.045,Z 365.047,A -85,B 0,C 180,E1 -8381.608,E2 -8381.608} C_VEL
LIN {X 0,Y 454.48,Z 356.866,A -85,B 0,C 180,E1 -8382.503,E2 -8382.503} C_VEL
LIN {X 0,Y 454.83,Z 348.3,A -85,B 0,C 180,E1 -8383.292,E2 -8383.292} C_VEL
LIN {X 0,Y 455.334,Z 339.634,A -85,B 0,C 180,E1 -8383.955,E2 -8383.955} C_VEL
LIN {X 0,Y 455.749,Z 330.881,A -85,B 0,C 180,E1 -8384.512,E2 -8384.512} C_VEL
LIN {X 0,Y 456.143,Z 322.368,A -85,B 0,C 180,E1 -8384.955,E2 -8384.955} C_VEL
LIN {X 0,Y 454.609,Z 311.023,A -85,B 0,C 180,E1 -8385.469,E2 -8385.469} C_VEL
LIN {X 0,Y 452.625,Z 300.052,A -85,B 0,C 180,E1 -8385.849,E2 -8385.849} C_VEL
LIN {X 0,Y 452.566,Z 299.42,A -85,B 0,C 180,E1 -8385.895,E2 -8385.895} C_VEL
LIN {X 0,Y 452.675,Z 293.603,A -85,B 0,C 180,E1 -8389.028,E2 -8389.028} C_VEL
LIN {X 0,Y 452.792,Z 288.501,A -85,B 0,C 180,E1 -8391.87,E2 -8391.87} C_VEL
LIN {X 0,Y 452.987,Z 283.443,A -85,B 0,C 180,E1 -8394.764,E2 -8394.764} C_VEL
LIN {X 0,Y 453.189,Z 278.192,A -85,B 0,C 180,E1 -8397.873,E2 -8397.873} C_VEL
LIN {X 0,Y 453.462,Z 273.503,A -85,B 0,C 180,E1 -8400.76,E2 -8400.76} C_VEL
LIN {X 0,Y 453.766,Z 268.646,A -85,B 0,C 180,E1 -8403.887,E2 -8403.887} C_VEL
LIN {X 0,Y 454.028,Z 263.876,A -85,B 0,C 180,E1 -8407.134,E2 -8407.134} C_VEL
LIN {X 0,Y 454.2,Z 260.747,A -85,B 0,C 180,E1 -8409.375,E2 -8409.375} C_VEL
LIN {X 0,Y 454.356,Z 257.238,A -85,B 0,C 180,E1 -8412.054,E2 -8412.054} C_VEL
LIN {X 0,Y 454.148,Z 254.144,A -85,B 0,C 180,E1 -8414.61,E2 -8414.61} C_VEL
LIN {X 0,Y 453.556,Z 250.182,A -85,B 0,C 180,E1 -8418.214,E2 -8418.214} C_VEL
LIN {X 0,Y 453.478,Z 249.499,A -85,B 0,C 180,E1 -8419.41,E2 -8419.41} C_VEL
LIN {X 0,Y 453.455,Z 249.502,A -85,B 0,C 180,E1 -8422.807,E2 -8422.807} C_VEL
LIN {X 0,Y 453.473,Z 249.502,A -85,B 0,C 180,E1 -8426.083,E2 -8426.083} C_VEL
LIN {X 0,Y 453.479,Z 249.494,A -85,B 0,C 180,E1 -8429.237,E2 -8429.237} C_VEL
LIN {X 0,Y 453.493,Z 249.495,A -85,B 0,C 180,E1 -8432.291,E2 -8432.291} C_VEL
LIN {X 0,Y 453.496,Z 249.493,A -85,B 0,C 180,E1 -8435.26,E2 -8435.26} C_VEL
LIN {X 0,Y 453.482,Z 249.494,A -85,B 0,C 180,E1 -8438.411,E2 -8438.411} C_VEL
LIN {X 0,Y 453.523,Z 249.488,A -85,B 0,C 180,E1 -8441.004,E2 -8441.004} C_VEL
LIN {X 0,Y 453.569,Z 249.487,A -85,B 0,C 180,E1 -8443.875,E2 -8443.875} C_VEL
LIN {X 0,Y 453.562,Z 249.49,A -85,B 0,C 180,E1 -8447.467,E2 -8447.467} C_VEL
LIN {X 0,Y 453.573,Z 249.485,A -85,B 0,C 180,E1 -8451.082,E2 -8451.082} C_VEL
LIN {X 0,Y 453.649,Z 249.475,A -85,B 0,C 180,E1 -8453.769,E2 -8453.769} C_VEL
LIN {X 0,Y 453.702,Z 249.473,A -85,B 0,C 180,E1 -8457.331,E2 -8457.331} C_VEL
LIN {X 0,Y 453.807,Z 249.453,A -85,B 0,C 180,E1 -8459.995,E2 -8459.995} C_VEL
LIN {X 0,Y 453.728,Z 249.464,A -85,B 0,C 180,E1 -8462.658,E2 -8462.658} C_VEL
LIN {X 0,Y 453.643,Z 249.473,A -85,B 0,C 180,E1 -8466.22,E2 -8466.22} C_VEL
LIN {X 0,Y 453.567,Z 249.489,A -85,B 0,C 180,E1 -8468.908,E2 -8468.908} C_VEL
LIN {X 0,Y 453.544,Z 249.488,A -85,B 0,C 180,E1 -8472.523,E2 -8472.523} C_VEL
LIN {X 0,Y 453.521,Z 249.489,A -85,B 0,C 180,E1 -8476.19,E2 -8476.19} C_VEL
LIN {X 0,Y 453.491,Z 249.496,A -85,B 0,C 180,E1 -8479.034,E2 -8479.034} C_VEL
LIN {X 0,Y 453.448,Z 249.497,A -85,B 0,C 180,E1 -8481.831,E2 -8481.831} C_VEL
LIN {X 0,Y 453.476,Z 249.5,A -85,B 0,C 180,E1 -8484.729,E2 -8484.729} C_VEL
LIN {X 0,Y 453.498,Z 249.492,A -85,B 0,C 180,E1 -8487.954,E2 -8487.954} C_VEL
LIN {X 0,Y 453.428,Z 249.5,A -85,B 0,C 180,E1 -8491.519,E2 -8491.519} C_VEL
LIN {X 0,Y 453.449,Z 249.5,A -85,B 0,C 180,E1 -8494.772,E2 -8494.772} C_VEL
LIN {X 0,Y 453.437,Z 249.506,A -85,B 0,C 180,E1 -8498.305,E2 -8498.305} C_VEL
LIN {X 0,Y 453.472,Z 249.497,A -85,B 0,C 180,E1 -8500.601,E2 -8500.601} C_VEL
LIN {X 0,Y 453.477,Z 249.501,A -85,B 0,C 180,E1 -8504.209,E2 -8504.209} C_VEL
LIN {X 0,Y 453.442,Z 249.498,A -85,B 0,C 180,E1 -8507.004,E2 -8507.004} C_VEL
LIN {X 0,Y 453.485,Z 249.494,A -85,B 0,C 180,E1 -8510.551,E2 -8510.551} C_VEL
LIN {X 0,Y 453.402,Z 249.511,A -85,B 0,C 180,E1 -8513.913,E2 -8513.913} C_VEL
LIN {X 0,Y 453.425,Z 249.501,A -85,B 0,C 180,E1 -8517.147,E2 -8517.147} C_VEL
LIN {X 0,Y 453.456,Z 249.498,A -85,B 0,C 180,E1 -8520.268,E2 -8520.268} C_VEL
LIN {X 0,Y 453.455,Z 249.499,A -85,B 0,C 180,E1 -8523.291,E2 -8523.291} C_VEL
LIN {X 0,Y 453.458,Z 249.497,A -85,B 0,C 180,E1 -8526.237,E2 -8526.237} C_VEL
LIN {X 0,Y 453.455,Z 249.499,A -85,B 0,C 180,E1 -8529.117,E2 -8529.117} C_VEL
LIN {X 0,Y 453.457,Z 249.501,A -85,B 0,C 180,E1 -8531.943,E2 -8531.943} C_VEL
LIN {X 0,Y 453.5,Z 249.495,A -85,B 0,C 180,E1 -8534.725,E2 -8534.725} C_VEL
LIN {X 0,Y 453.523,Z 249.49,A -85,B 0,C 180,E1 -8538.378,E2 -8538.378} C_VEL
LIN {X 0,Y 453.591,Z 249.484,A -85,B 0,C 180,E1 -8541.984,E2 -8541.984} C_VEL
LIN {X 0,Y 453.585,Z 249.485,A -85,B 0,C 180,E1 -8543.062,E2 -8543.062} C_VEL
LIN {X 0,Y 452.9,Z 249.571,A -85,B 0,C 180,E1 -8543.803,E2 -8543.803} C_VEL
